PROPERTY PUBLIC classHintActive : BOOL
GET
classHintActive													:= ClassInfo[TCEVENTCLASS_HINT] <> 0;
END_GET
END_PROPERTY

PROPERTY PUBLIC classInstructionActive : BOOL
GET
classInstructionActive													:= ClassInfo[TCEVENTCLASS_INSTRUCTION] <> 0;
END_GET
END_PROPERTY

PROPERTY PUBLIC classMaintenanceActive : BOOL
GET
classMaintenanceActive													:= ClassInfo[TCEVENTCLASS_MAINTENANCE] <> 0;
END_GET
END_PROPERTY

PROPERTY PUBLIC classMessageActive : BOOL
GET
classMessageActive													:= ClassInfo[TCEVENTCLASS_MESSAGE] <> 0;
END_GET
END_PROPERTY

PROPERTY PUBLIC classNoneActive : BOOL
GET
ClassNoneActive													:= ClassInfo[TCEVENTCLASS_NONE] <> 0;
END_GET
END_PROPERTY

PROPERTY PUBLIC classParamErrorActive : BOOL
GET
ClassParamErrorActive													:= ClassInfo[TCEVENTCLASS_PARAMERROR] <> 0;
END_GET
END_PROPERTY

PROPERTY PUBLIC classStateinfoActive : BOOL
GET
ClassStateinfoActive													:= ClassInfo[TCEVENTCLASS_STATEINFO] <> 0;
END_GET
END_PROPERTY

PROPERTY PUBLIC classWarningActive : BOOL
GET
ClassWarningActive													:= ClassInfo[TCEVENTCLASS_WARNING] <> 0;
END_GET
END_PROPERTY

METHOD PUBLIC clear : BOOL //Return value = TRUE if execution finished 
VAR_INPUT
END_VAR
	MEMSET(ADR(ClassInfo),0,SIZEOF(ClassInfo));
	MEMSET(ADR(PriorityInfo),0,SIZEOF(PriorityInfo));
	NoOfQuitRequiredEvents									:= 0;	
	NoOfActiveEvents										:= 0;
	Clear													:= TRUE;
END_METHOD

{attribute 'hide'}
METHOD PUBLIC countIn : BOOL //Return value = TRUE if execution finished 
VAR_IN_OUT
	Status													:	DWORD; (*	.0 - .8 = event of <class id> is active / .15 confirm required / .16 = Level 0 , .17 = Level 1 , .18 = Level 2, ..........
																			TCEVENTCLASS_NONE			:=0,	(* No class *)
																			TCEVENTCLASS_MAINTENANCE	:=1,	(* Maintenance hint *)
																			TCEVENTCLASS_MESSAGE		:=2,	(* Message *)
																			TCEVENTCLASS_HINT			:=3,	(* Hint *)
																			TCEVENTCLASS_STATEINFO		:=4,	(* State information *)
																			TCEVENTCLASS_INSTRUCTION	:=5,	(* Instruction *)
																			TCEVENTCLASS_WARNING		:=6,	(* Warning *)
																			TCEVENTCLASS_ALARM			:=7,	(* Alarm *)
																			TCEVENTCLASS_PARAMERROR		:=8		(* Parameter error *)  *)
END_VAR
IF TestAndSet(TaskInterlockCountIn)
THEN
	IF Status.0 THEN ClassInfo[TCEVENTCLASS_NONE] 				:= ClassInfo[TCEVENTCLASS_NONE] + 1; 									
	ELSIF Status.1 THEN ClassInfo[TCEVENTCLASS_MAINTENANCE] 	:= ClassInfo[TCEVENTCLASS_MAINTENANCE] + 1; 
	ELSIF Status.2 THEN ClassInfo[TCEVENTCLASS_MESSAGE] 		:= ClassInfo[TCEVENTCLASS_MESSAGE] + 1; 	
	ELSIF Status.3 THEN ClassInfo[TCEVENTCLASS_HINT] 			:= ClassInfo[TCEVENTCLASS_HINT] + 1; 		
	ELSIF Status.4 THEN ClassInfo[TCEVENTCLASS_STATEINFO] 		:= ClassInfo[TCEVENTCLASS_STATEINFO] + 1; 	
	ELSIF Status.5 THEN ClassInfo[TCEVENTCLASS_INSTRUCTION] 	:= ClassInfo[TCEVENTCLASS_INSTRUCTION] + 1; 
	ELSIF Status.6 THEN ClassInfo[TCEVENTCLASS_WARNING] 		:= ClassInfo[TCEVENTCLASS_WARNING] + 1; 	
	ELSIF Status.7 THEN ClassInfo[TCEVENTCLASS_ALARM] 			:= ClassInfo[TCEVENTCLASS_ALARM] + 1; 		
	ELSIF Status.8 THEN ClassInfo[TCEVENTCLASS_PARAMERROR] 		:= ClassInfo[TCEVENTCLASS_PARAMERROR] + 1; 	
	END_IF
	
	IF Status.15 THEN NoOfQuitRequiredEvents 					:= NoOfQuitRequiredEvents + 1; END_IF
	
	IF status.16 THEN PriorityInfo[0]							:= PriorityInfo[0] + 1;						
	ELSIF status.17 THEN PriorityInfo[1]						:= PriorityInfo[1] + 1	;						
	ELSIF status.18 THEN PriorityInfo[2]						:= PriorityInfo[2] + 1;						
	ELSIF status.19 THEN PriorityInfo[3]						:= PriorityInfo[3] + 1;						
	ELSIF status.20 THEN PriorityInfo[4]						:= PriorityInfo[4] + 1;						
	ELSIF status.21 THEN PriorityInfo[5]						:= PriorityInfo[5] + 1;						
	ELSIF status.22 THEN PriorityInfo[6]						:= PriorityInfo[6] + 1;						
	ELSIF status.23 THEN PriorityInfo[7]						:= PriorityInfo[7] + 1	;						
	END_IF
	
	//set active flag	
	NoOfActiveEvents											:= NoOfActiveEvents + 1;
	
	status.31 													:= TRUE; 
	CountIn														:= TRUE;
	TaskInterlockCountIn										:= FALSE;
END_IF
END_METHOD

// {attribute 'hide'}
METHOD PUBLIC countOut : BOOL //Return value = TRUE if execution finished 
VAR_IN_OUT
	Status													:	DWORD; (*	.0 - .8 = event of <class id> is active / .15 confirm required / .16 = Level 0 , .17 = Level 1 , .18 = Level 2, ..........
																			TCEVENTCLASS_NONE			:=0,	(* No class *)
																			TCEVENTCLASS_MAINTENANCE	:=1,	(* Maintenance hint *)
																			TCEVENTCLASS_MESSAGE		:=2,	(* Message *)
																			TCEVENTCLASS_HINT			:=3,	(* Hint *)
																			TCEVENTCLASS_STATEINFO		:=4,	(* State information *)
																			TCEVENTCLASS_INSTRUCTION	:=5,	(* Instruction *)
																			TCEVENTCLASS_WARNING		:=6,	(* Warning *)
																			TCEVENTCLASS_ALARM			:=7,	(* Alarm *)
																			TCEVENTCLASS_PARAMERROR		:=8		(* Parameter error *)  *)
END_VAR
IF TestAndSet(TaskInterlockCountOut)
THEN
	IF Status.0 THEN ClassInfo[TCEVENTCLASS_NONE] 				:= MAX(0,ClassInfo[TCEVENTCLASS_NONE] - 1); 		
	ELSIF Status.1 THEN ClassInfo[TCEVENTCLASS_MAINTENANCE] 	:= MAX(0,ClassInfo[TCEVENTCLASS_MAINTENANCE] - 1);	
	ELSIF Status.2 THEN ClassInfo[TCEVENTCLASS_MESSAGE] 		:= MAX(0,ClassInfo[TCEVENTCLASS_MESSAGE] - 1); 		
	ELSIF Status.3 THEN ClassInfo[TCEVENTCLASS_HINT] 			:= MAX(0,ClassInfo[TCEVENTCLASS_HINT] - 1); 		
	ELSIF Status.4 THEN ClassInfo[TCEVENTCLASS_STATEINFO] 		:= MAX(0,ClassInfo[TCEVENTCLASS_STATEINFO] - 1); 	
	ELSIF Status.5 THEN ClassInfo[TCEVENTCLASS_INSTRUCTION] 	:= MAX(0,ClassInfo[TCEVENTCLASS_INSTRUCTION] - 1);	
	ELSIF Status.6 THEN ClassInfo[TCEVENTCLASS_WARNING] 		:= MAX(0,ClassInfo[TCEVENTCLASS_WARNING] - 1); 	
	ELSIF Status.7 THEN ClassInfo[TCEVENTCLASS_ALARM] 			:= MAX(0,ClassInfo[TCEVENTCLASS_ALARM] - 1); 		
	ELSIF Status.8 THEN ClassInfo[TCEVENTCLASS_PARAMERROR] 		:= MAX(0,ClassInfo[TCEVENTCLASS_PARAMERROR] - 1); 	
	END_IF
																	  
	IF Status.15 THEN NoOfQuitRequiredEvents 					:=  MAX(0,NoOfQuitRequiredEvents - 1); 	
	END_IF
																	   
	IF status.16 THEN PriorityInfo[0]							:=  MAX(0,PriorityInfo[0] - 1);						
	ELSIF status.17 THEN PriorityInfo[1]						:=  MAX(0,PriorityInfo[1] - 1);						
	ELSIF status.18 THEN PriorityInfo[2]						:=  MAX(0,PriorityInfo[2] - 1);						
	ELSIF status.19 THEN PriorityInfo[3]						:=  MAX(0,PriorityInfo[3] - 1);						
	ELSIF status.20 THEN PriorityInfo[4]						:=  MAX(0,PriorityInfo[4] - 1);						
	ELSIF status.21 THEN PriorityInfo[5]						:=  MAX(0,PriorityInfo[5] - 1);						
	ELSIF status.22 THEN PriorityInfo[6]						:=  MAX(0,PriorityInfo[6] - 1);						
	ELSIF status.23 THEN PriorityInfo[7]						:=  MAX(0,PriorityInfo[7] - 1);						
	END_IF
	
	NoOfActiveEvents											:= MAX(0,NoOfActiveEvents - 1);
	status.31													:= FALSE; //Active flag reset
	CountOut													:= TRUE;
	TaskInterlockCountOut										:= FALSE;
END_IF
END_METHOD

METHOD INTERNAL initEvent : DWORD //Return status 
VAR_IN_OUT
	SetClass								:	E_TcEventClass;
	EventConfig								:	TcEvent;
END_VAR
		(* Event Config *)
		InitEvent											:= 0;
		IF SetClass = TC2_SYSTEM.TCEVENTCLASS_NONE 				
		THEN	
			EventConfig.Class								:= SetClass;
			EventConfig.bQuitRequired						:= PARAM.EVENT_HANDLING_CONFIG.CLASS_NONE_QUIT_REQUIRED;
			InitEvent.15									:= PARAM.EVENT_HANDLING_CONFIG.CLASS_NONE_QUIT_REQUIRED;
			EventConfig.Prio								:= PARAM.EVENT_HANDLING_CONFIG.CLASS_NONE_PRIORITY;
			InitEvent										:= SETBIT32(InitEvent,TO_SINT(PARAM.EVENT_HANDLING_CONFIG.CLASS_NONE_PRIORITY) + 16);	
			InitEvent.0										:= TRUE;													
			
		ELSIF SetClass = TC2_SYSTEM.TCEVENTCLASS_MAINTENANCE 
		THEN
			EventConfig.Class								:= SetClass;
			EventConfig.bQuitRequired						:= PARAM.EVENT_HANDLING_CONFIG.CLASS_MAINTENANCE_QUIT_REQUIRED;
			InitEvent.15									:= PARAM.EVENT_HANDLING_CONFIG.CLASS_MAINTENANCE_QUIT_REQUIRED;
			EventConfig.Prio								:= PARAM.EVENT_HANDLING_CONFIG.CLASS_MAINTENANCE_PRIORITY;
			InitEvent										:= SETBIT32(InitEvent,TO_SINT(PARAM.EVENT_HANDLING_CONFIG.CLASS_MAINTENANCE_PRIORITY) + 16);
			InitEvent.1										:= TRUE;
		ELSIF SetClass = TC2_SYSTEM.TCEVENTCLASS_MESSAGE 		
		THEN
			EventConfig.Class								:= SetClass;
			EventConfig.bQuitRequired						:= PARAM.EVENT_HANDLING_CONFIG.CLASS_MESSAGE_QUIT_REQUIRED;
			InitEvent.15									:= PARAM.EVENT_HANDLING_CONFIG.CLASS_MESSAGE_QUIT_REQUIRED;
			EventConfig.Prio								:= PARAM.EVENT_HANDLING_CONFIG.CLASS_MESSAGE_PRIORITY;
			InitEvent										:= SETBIT32(InitEvent,TO_SINT(PARAM.EVENT_HANDLING_CONFIG.CLASS_MESSAGE_PRIORITY) + 16);
			InitEvent.2										:= TRUE;
		ELSIF SetClass = TC2_SYSTEM.TCEVENTCLASS_HINT 			
		THEN
			EventConfig.Class								:= SetClass;
			EventConfig.bQuitRequired						:= PARAM.EVENT_HANDLING_CONFIG.CLASS_HINT_QUIT_REQUIRED;
			InitEvent.15									:= PARAM.EVENT_HANDLING_CONFIG.CLASS_HINT_QUIT_REQUIRED;
			EventConfig.Prio								:= PARAM.EVENT_HANDLING_CONFIG.CLASS_HINT_PRIORITY;
			InitEvent										:= SETBIT32(InitEvent,TO_SINT(PARAM.EVENT_HANDLING_CONFIG.CLASS_HINT_PRIORITY) + 16);
			InitEvent.3										:= TRUE;
		ELSIF SetClass = TC2_SYSTEM.TCEVENTCLASS_STATEINFO 	
		THEN
			EventConfig.Class								:= SetClass;
			EventConfig.bQuitRequired						:= PARAM.EVENT_HANDLING_CONFIG.CLASS_STATEINFO_QUIT_REQUIRED;
			InitEvent.15									:= PARAM.EVENT_HANDLING_CONFIG.CLASS_STATEINFO_QUIT_REQUIRED;
			EventConfig.Prio								:= PARAM.EVENT_HANDLING_CONFIG.CLASS_STATEINFO_PRIORITY;
			InitEvent										:= SETBIT32(InitEvent,TO_SINT(PARAM.EVENT_HANDLING_CONFIG.CLASS_STATEINFO_PRIORITY) + 16);
			InitEvent.4										:= TRUE;
		ELSIF SetClass = TC2_SYSTEM.TCEVENTCLASS_INSTRUCTION 
		THEN
			EventConfig.Class								:= SetClass;
			EventConfig.bQuitRequired						:= PARAM.EVENT_HANDLING_CONFIG.CLASS_INSTRUCTION_QUIT_REQUIRED;
			InitEvent.15									:= PARAM.EVENT_HANDLING_CONFIG.CLASS_INSTRUCTION_QUIT_REQUIRED;
			EventConfig.Prio								:= PARAM.EVENT_HANDLING_CONFIG.CLASS_INSTRUCTION_PRIORITY;
			InitEvent										:= SETBIT32(InitEvent,TO_SINT(PARAM.EVENT_HANDLING_CONFIG.CLASS_INSTRUCTION_PRIORITY) + 16);
			InitEvent.5										:= TRUE;
		ELSIF SetClass = TC2_SYSTEM.TCEVENTCLASS_WARNING 		
		THEN
			EventConfig.Class								:= SetClass;
			EventConfig.bQuitRequired						:= PARAM.EVENT_HANDLING_CONFIG.CLASS_WARNING_QUIT_REQUIRED;
			InitEvent.15									:= PARAM.EVENT_HANDLING_CONFIG.CLASS_WARNING_QUIT_REQUIRED;
			EventConfig.Prio								:= PARAM.EVENT_HANDLING_CONFIG.CLASS_WARNING_PRIORITY;
			InitEvent										:= SETBIT32(InitEvent,TO_SINT(PARAM.EVENT_HANDLING_CONFIG.CLASS_WARNING_PRIORITY) + 16);
			InitEvent.6										:= TRUE;
		ELSIF SetClass = TC2_SYSTEM.TCEVENTCLASS_ALARM 		
		THEN
			EventConfig.Class								:= SetClass;
			EventConfig.bQuitRequired						:= PARAM.EVENT_HANDLING_CONFIG.CLASS_ALARM_QUIT_REQUIRED;
			InitEvent.15									:= PARAM.EVENT_HANDLING_CONFIG.CLASS_ALARM_QUIT_REQUIRED;
			EventConfig.Prio								:= PARAM.EVENT_HANDLING_CONFIG.CLASS_ALARM_PRIORITY;
			InitEvent										:= SETBIT32(InitEvent,TO_SINT(PARAM.EVENT_HANDLING_CONFIG.CLASS_ALARM_PRIORITY) + 16);
			InitEvent.7										:= TRUE;
		ELSIF SetClass = TC2_SYSTEM.TCEVENTCLASS_PARAMERROR 	
		THEN
			EventConfig.Class								:= SetClass;
			EventConfig.bQuitRequired						:= PARAM.EVENT_HANDLING_CONFIG.CLASS_PARAMERROR_QUIT_REQUIRED;
			InitEvent.15									:= PARAM.EVENT_HANDLING_CONFIG.CLASS_PARAMERROR_QUIT_REQUIRED;
			EventConfig.Prio								:= PARAM.EVENT_HANDLING_CONFIG.CLASS_PARAMERROR_PRIORITY;
			InitEvent										:= SETBIT32(InitEvent,TO_SINT(PARAM.EVENT_HANDLING_CONFIG.CLASS_PARAMERROR_PRIORITY) + 16);
			InitEvent.8										:= TRUE;
		ELSE 
			EventConfig.Class								:= SetClass;
			EventConfig.bQuitRequired						:= PARAM.EVENT_HANDLING_CONFIG.CLASS_ALARM_QUIT_REQUIRED;
			InitEvent.15									:= PARAM.EVENT_HANDLING_CONFIG.CLASS_ALARM_QUIT_REQUIRED;
			EventConfig.Prio								:= PARAM.EVENT_HANDLING_CONFIG.CLASS_ALARM_PRIORITY;
			InitEvent										:= SETBIT32(InitEvent,TO_SINT(PARAM.EVENT_HANDLING_CONFIG.CLASS_ALARM_PRIORITY) + 16);
			InitEvent.7										:= TRUE;
		END_IF
END_METHOD

METHOD PUBLIC isClassActive : BOOL  //Return value = TRUE if EventClass is currently active
VAR_INPUT
	TcEventClass											:	E_TcEventClass;
END_VAR
IF TcEventClass < MIN_CLASS OR TcEventClass > MAX_CLASS
THEN
	IsClassActive											:= TRUE;
ELSE
	IsClassActive											:= ClassInfo[TcEventClass] <> 0;
END_IF
END_METHOD

PROPERTY PUBLIC isConfirmReqActive : BOOL
GET
isConfirmReqActive											:= NoOfQuitRequiredEvents <> 0;
END_GET
END_PROPERTY

METHOD PUBLIC isPriorityActive : BOOL //Return value = TRUE if priority is active
VAR_INPUT
	IN														:	INT;
END_VAR
IF IN < MIN_PRIORITY OR IN > MAX_PRIORITY
THEN
	IsPriorityActive										:= TRUE;
ELSE
	IsPriorityActive										:= PriorityInfo[In] <> 0;
END_IF
END_METHOD

END_FUNCTION_BLOCK

// POUs/EventLogger/EventsWriteToLogbook
{attribute 'no_check'}
//Write new event logger messages from "ReadAdsEvent" instance into "LogBook" instance
FUNCTION_BLOCK EventsWriteToLogbook
VAR_OUTPUT CONSTANT
{attribute 'displaymode':='binary'}
	OPTION_ADD_DT_TO_MSG_STRING								:	BYTE := 2#0000_0001;
{attribute 'displaymode':='binary'}
	OPTION_ADD_CLASS_TO_MSG_STRING							:	BYTE := 2#0000_0010;
{attribute 'displaymode':='binary'}
	OPTION_ADD_SOURCE_TO_MSG_STRING							:	BYTE := 2#0000_0100;	//Default option
{attribute 'displaymode':='binary'}
	OPTION_ADD_SOURCE_ID_TO_MSG_STRING						:	BYTE := 2#0000_1000; 
{attribute 'displaymode':='binary'}
	OPTION_ADD_MSG_ID_TO_MSG_STRING							:	BYTE := 2#0001_0000;	//Default option	
{attribute 'displaymode':='binary'}
	OPTION_ADD_MSG_DT_TO_LOGBOOK_TIMESTAMP					:	BYTE := 2#0010_0000;	
{attribute 'displaymode':='binary'}
	OPTION_ADD_MSG_STATE_ID_TO_MSG_STRING					:	BYTE := 2#0100_0000;	//Add event state before text
END_VAR
VAR_INPUT
	Enable													:	BOOL	:= FALSE;	//Activate the function block
{attribute 'displaymode':='binary'}
	Options													:	BYTE 	:= OPTION_ADD_SOURCE_TO_MSG_STRING OR OPTION_ADD_MSG_ID_TO_MSG_STRING;
END_VAR                                                     
VAR_IN_OUT                                                  
	EventlogRead											:	EventlogRead;		//ReadAdsEvent instance
	LogBook													:	LogBook_wEventClass;//Logbook instance 
END_VAR                                                     
VAR_OUTPUT                                                  
	LastEventDT												:	DT;					//Date and time of last checked event
END_VAR                                                         			
VAR
(* Memory ******************************************************)
	LastEntryTimestamp										:	T_DCTIME64;			//Date of last event in this cycle
	LastEventTimestamp										:	T_DCTIME64;			//Timestamp of last added event
	ExitMarker												:	BOOL;
	MemLogbookOptions										:	BYTE;	
	MemClass												:	E_TcEventClass := TC2_SYSTEM.TCEVENTCLASS_ALARM;
	MemTimestamp											:	TIMESTRUCT;
	LenMem													:	INT;

	
(* Timer *******************************************************)

(* Trigger *****************************************************)

(* Blocks ******************************************************)

(* Error *******************************************************)

(* Dummys ******************************************************)
	i														: 	INT := 0; 
	k,j														:	INT;
	OK														:	BOOL;
END_VAR

(* Read new events and write into logbook 							*)
(********************************************************************)

(* action ***********************************************************)
IF Enable 
THEN
	IF EventlogRead.Done
	THEN //Start read events
	
		//first save Logbook settings 
		MemTimestamp										:= LogBook.Timestamp;
		MemLogbookOptions									:= LogBook.Options;		
		MemClass											:= LogBook.eClass;
	(*	LogBook.Options										:= LogBook.Options 
																AND Logbook.OPTION_WRITE_TO_ADSLOG AND Logbook.OPTION_WRITE_TO_FILE 
																AND Logbook.OPTION_ADD_TIME_TO_MSG_STRING AND Logbook.OPTION_ADD_TIME_TO_MSG_STRING ; *)
		
		//Check list for new entrys
		ExitMarker											:= FALSE;
		FOR i := EventlogRead.TotalNumberOfEvents TO EventlogRead.MIN_EVENT BY - 1  
		DO
			IF EventlogRead.Event[i].Timestamp > LastEntryTimestamp
			THEN //New entries
				IF NOT ExitMarker 
					OR //Events with event newer timestamp, exit and continue at next cycle
					EventlogRead.Event[i].Timestamp = LastEventTimestamp
				THEN //new message
					ExitMarker								:= TRUE;
					LastEventTimestamp						:= EventlogRead.Event[i].Timestamp;
										
					IF _formatMsg(EventlogRead.LangId, EventlogRead.Event[i], LogBook)
					THEN //Write message to logbook	
						Logbook();
					END_IF
					
				ELSE //add messages the next time
					EXIT; 
				END_IF
				
			ELSE //old messages
				;
			END_IF
		
		END_FOR		
		
		//Record timestamp of last event
		LastEntryTimestamp									:= LastEventTimestamp;

		//Recover old entries	
		LogBook.Options										:= MemLogbookOptions;
		LogBook.eClass										:= MemClass;
		LogBook.Timestamp									:= MemTimestamp;				
	END_IF	
END_IF

(*******************************************************************************)

METHOD PROTECTED _formatMsg : BOOL
VAR_INPUT
	Lcid													:	eLCID;
END_VAR
VAR_IN_OUT
	Event													 : EVENTLOG_READ_DATA;
	LogBook													:	LogBook_wEventClass;//Logbook instance 
END_VAR
//2020-05-30-07:06:08.436;<EventClass txt>;<Source ID>;<Event Id>;<Event state>;CoE Drive | AxisY - Remote control over fieldbus not active  	

	//Add class to log book entry
	LogBook.eClass											:= Event.eClass;	
	Logbook.Msg												:= '';
	
	//Event timestamp to logbook timestamp
	IF OPtions.5
	THEN
		LogBook.Timestamp 									:= DT_TO_SYSTEMTIME(Event.TimestampDT);			
	END_IF
	
	//add date and time
	IF Options.0
	THEN					
		LogBook.Msg											:= DT_TO_STRING(Event.TimestampDT);			
		LogBook.Msg											:= DELETE(LogBook.Msg, 3, 1); //delete DT# 
		LogBook.Msg 										:= CONCAT(LogBook.Msg,';');					
	END_IF
		
	//add event class
	IF Options.1
	THEN
		LogBook.Msg											:= CONCAT(LogBook.Msg,GetEventClassText(Event.eClass));
		LogBook.Msg 										:= CONCAT(LogBook.Msg,';');
	END_IF

	//add source id 
	IF Options.3 
	THEN
		LogBook.Msg 										:= CONCAT(LogBook.Msg,TO_STRING(Event.Sourceid));
		LogBook.Msg 										:= CONCAT(LogBook.Msg,';');		
	END_IF							
							
	//add event id 
	IF Options.4
	THEN
		LogBook.Msg 										:= CONCAT(LogBook.Msg,DWORD_TO_STRING(Event.id));
		LogBook.Msg 										:= CONCAT(LogBook.Msg,';');				
	END_IF					
	
	//add event state
	IF Options.6
	THEN
		LogBook.Msg 										:= CONCAT(LogBook.Msg,DWORD_TO_STRING(Event.State));
		LogBook.Msg 										:= CONCAT(LogBook.Msg,';');				
	END_IF					

	//add event source text
	IF Options.2
	THEN
		IF Lcid <> eLCID.CN
		THEN
			LogBook.Msg 									:= CONCAT(LogBook.Msg,WSTRING_TO_STRING(Event.Source));
			LogBook.Msg 									:= CONCAT(LogBook.Msg,' | ');	
		ELSIF NOT Options.3    
		THEN                               
			LogBook.Msg 									:= CONCAT(LogBook.Msg,CONCAT('Source Id[', UDINT_TO_STRING(Event.Sourceid)));
			LogBook.Msg 									:= CONCAT(LogBook.Msg,'] | ');								
		END_IF	
	END_IF
		
	IF Lcid <> eLCID.CN
	THEN
		LogBook.Msg											:= CONCAT(LogBook.Msg,WSTRING_TO_STRING(Event.MsgText));
	ELSE
		LogBook.Msg 										:= CONCAT(LogBook.Msg, SEL(Options.4 , CONCAT('EventId[' ,CONCAT(UDINT_TO_STRING(Event.id),'] <Unicode active>')) , '<Unicode active>'));										
	END_IF

	_formatMsg												:= TRUE;
	
(**********************************************************************************************)
END_METHOD

END_FUNCTION_BLOCK

// POUs/Logging/Logbook
{attribute 'no_check'}
//PLC Logbook for debugging, records a number of "MAX_DATA" messages with timestamp.
//The Logbook Puplisher can be used to forward messages from the logbook to several subscriber (Write into Logfile, display via EventLogger, send to Syslog Server)
//
//Parameter Timestamp needs to be updated externaly every cycle if needed
//
//Function "LogWithEventClass" is used inside
FUNCTION_BLOCK Logbook IMPLEMENTS I_Logbook                 									
VAR_OUTPUT CONSTANT     									
//Parameter
	MIN_DATA												:	INT := 1;
	MAX_DATA												:	INT := PARAM.LOGBOOK_MAX_DATA; //see library parameter to customize parameter	
                        									
//option settings to modify the message string and behavior
{attribute 'displaymode':='binary'}
	OPTION_WRITE_TO_ADSLOG									: 	BYTE :=2#0000_0100; //Write entry directly to TwinCAT logger (shown in XAE output)
{attribute 'displaymode':='binary'}
	OPTION_ADD_TIME_TO_MSG_STRING							: 	BYTE :=2#0000_1000;	//Add time stamp to message string 
{attribute 'displaymode':='binary'}
	OPTION_ADD_DATE_TO_MSG_STRING							: 	BYTE :=2#0001_0000; //Add date to message string
END_VAR                 									
VAR_INPUT               									                       		
{attribute 'displaymode':='binary'}
	Options													:	BYTE := 2#0000_0000;			(* option constants are alreay predefined, so they can accordingly be passed symbolically to the block
																								Bit 0 = 
																								Bit 1 = 
																								Bit 2 = Send to TC Ads-Logger
																								Bit 3 = Add time to message string
																								Bit 4 = Add date to message string
																								Bit 5 = 
																								Bit 6 = 
														 										Bit 7 =  								
																								*)
                        									
// InputData         	
	Timestamp												:	TIMESTRUCT; //Time stamp need to be updated cylic if it will be used
	Msg														:	STRING(PARAM.LOGBOOK_MAX_MSG_STRING_LENGHT) := ''; //Message string which will written into the DataMsg array by executing the Fb																							
END_VAR             										
VAR_OUTPUT
	Data													:	ARRAY[MIN_DATA..MAX_DATA] OF LogbookData; // Recorded messages data
	CntAddedMessages										:	INT;
END_VAR
VAR
	TaskInterlock											:	BOOL;
END_VAR

(* LogBook 									 *)
(*********************************************)

(* call method *********************************************)
	_Write(Msg);
(***********************************************************)

METHOD PROTECTED _write : BOOL
VAR_IN_OUT
	Msg														:	STRING(PARAM.LOGBOOK_MAX_MSG_STRING_LENGHT);
END_VAR
(* Write entry with every call ******************************)
IF LEN(MSG) = 0
THEN
	_Write													:= FALSE;
	RETURN;
ELSIF TestAndSet(TaskInterlock)
THEN	
	MEMMOVE(ADR(Data[MIN(MIN_DATA + 1,MAX_DATA)]), 	ADR(Data), 	SIZEOF(Data) - SIZEOF(Data[MIN_DATA]));
	
	(* Datensatz oben eintragen *)
	IF NOT Options.3 AND NOT Options.4
	THEN
		Data[MIN_DATA].Msg									:= Msg;
	ELSIF Options.3 AND Options.4              
	THEN                                                    
		Data[MIN_DATA].Msg									:= SYSTEMTIME_TO_STRING(Timestamp);
		Data[MIN_DATA].Msg									:= CONCAT(Data[MIN_DATA].Msg, ' | ');
		Data[MIN_DATA].Msg									:= CONCAT(Data[MIN_DATA].Msg, Msg);
	ELSIF Options.4                                   
	THEN                                                    
		Data[MIN_DATA].Msg									:= SYSTEMTIME_TO_STRING(Timestamp);
		Data[MIN_DATA].Msg									:=	MID(Data[MIN_DATA].Msg, 12 , 12);
		Data[MIN_DATA].Msg									:= CONCAT(Data[MIN_DATA].Msg, ' | ');
		Data[MIN_DATA].Msg									:= CONCAT(Data[MIN_DATA].Msg, Msg);
                                                            
	ELSE (* Only Date to Msg String *)                      
		Data[MIN_DATA].Msg									:= SYSTEMTIME_TO_STRING(Timestamp);
		Data[MIN_DATA].Msg									:= MID(Data[MIN_DATA].Msg, 8 , 3);
		Data[MIN_DATA].Msg									:= CONCAT(Data[MIN_DATA].Msg, ' | ');
		Data[MIN_DATA].Msg									:= CONCAT(Data[MIN_DATA].Msg, Msg);
	END_IF                                                  

	//Coyp current options from logbook into message	                                                        
	Data[MIN_DATA].Options									:= TO_WORD(Options);
		
	//Store time stamp
	Data[MIN_DATA].Timestamp								:= Timestamp;
	
	CntAddedMessages										:= MIN(MAX_DATA, CntAddedMessages + 1); 
	_Write													:= TRUE;
	TaskInterlock											:= FALSE;
END_IF

(************************************************************)
END_METHOD

METHOD PUBLIC delete : BOOL //Return value = TRUE if execution finished
VAR_INPUT
END_VAR

CntAddedMessages											:= 0;
MEMSET(ADR(Data),0,SIZEOF(Data));
delete														:= TRUE;
END_METHOD

METHOD PUBLIC getOldestMsg : BOOL //Return value TRUE = if finished successful -> new message read
VAR_IN_OUT
	data													: LogbookData;								
END_VAR
IF CntAddedMessages >= MIN_DATA AND CntAddedMessages <= MAX_DATA
	AND NOT TaskInterlock
THEN
	data													:= THIS^.Data[CntAddedMessages];
	THIS^.Data[CntAddedMessages].Options.15					:= FALSE; //New message
	CntAddedMessages										:= CntAddedMessages - 1;
	getOldestMsg											:= TRUE;
ELSE
	getOldestMsg											:= FALSE;
END_IF
END_METHOD

PROPERTY PUBLIC optAddDateToMsgText : BOOL
GET
optAddDateToMsgText := Options.4;
END_GET
SET
Options.4 := optAddDateToMsgText;
END_SET
END_PROPERTY

PROPERTY PUBLIC optAddTimeToMsgText : BOOL
GET
optAddTimeToMsgText := Options.3;
END_GET
SET
Options.3 := optAddTimeToMsgText;
END_SET
END_PROPERTY

PROPERTY Public optWiteEntryToTcAdsLogger : BOOL
GET
optWiteEntryToTcAdsLogger := Options.2;
END_GET
SET
Options.2 := optWiteEntryToTcAdsLogger;
END_SET
END_PROPERTY

{attribute 'monitoring' := 'call'}
PROPERTY PUBLIC rCntAddedMessages : Reference to INT //Reference to variable showing no of added messages (Counter will be decreased by getOldestMsg)
GET
rCntAddedMessages REF= CntAddedMessages;
END_GET
END_PROPERTY

METHOD PUBLIC readMsg : REFERENCE TO LogbookData //Return value is a REFERENCE to the by Index selected entry.  
VAR_INPUT
	Index											:	INT;						
END_VAR

readMsg													REF= THIS^.Data[LIMIT(MIN_DATA,Index,MAX_DATA)];
END_METHOD

METHOD PUBLIC write : BOOL //Return value = TRUE if execution finished
VAR_INPUT
	Msg														:	STRING(PARAM.LOGBOOK_MAX_MSG_STRING_LENGHT);
END_VAR

write														:= _Write(Msg);
IF options.2 
THEN
	write 													:= write AND 0 = adsLogHint(Msg, '');
END_IF
END_METHOD

END_FUNCTION_BLOCK

// POUs/Logging/I_Logbook
INTERFACE I_Logbook Extends __System.IQueryInterface

METHOD PUBLIC delete : BOOL //Return value = TRUE if execution finished
VAR_INPUT
END_VAR
END_METHOD

METHOD PUBLIC getOldestMsg : BOOL //Return value TRUE = if finished successful -> new message flag of entry will be reset
VAR_IN_OUT
	data													: LogbookData;								
END_VAR
END_METHOD

{attribute 'monitoring' := 'call'}
PROPERTY PUBLIC rCntAddedMessages : Reference to INT
GET
END_GET
END_PROPERTY

METHOD PUBLIC readMsg : REFERENCE TO LogbookData //Return value is a REFERENCE to the by Index selected entry.  
VAR_INPUT
	Index											:	INT;						
END_VAR
END_METHOD

METHOD PUBLIC write : BOOL //Return value = TRUE if execution finished
VAR_INPUT
	Msg														:	STRING(PARAM.LOGBOOK_MAX_MSG_STRING_LENGHT);
END_VAR
END_METHOD

END_INTERFACE

// POUs/Logging/Logbook_wEventClass
{attribute 'no_check'}
FUNCTION_BLOCK Logbook_wEventClass EXTENDS Logbook             									
VAR_OUTPUT CONSTANT     									
END_VAR                 									
VAR_INPUT               									                       		
	eClass													:	E_TcEventClass := TC2_SYSTEM.TCEVENTCLASS_NONE; //Possible event class for the entry																							
END_VAR             										
VAR_OUTPUT
END_VAR
VAR

END_VAR

(* LogBook 									 *)
(*********************************************)

(* call method *********************************************)
	Write(Msg);
(***********************************************************)

METHOD PUBLIC getClassFromOption : E_TcEventClass
VAR_INPUT
	Msgidx														:	INT;
END_VAR
IF Msgidx >= MIN_DATA AND Msgidx <= MAX_DATA
THEN
	GetClassFromOption.0 										:= Data[Msgidx].Options.8;
	GetClassFromOption.1 										:= Data[Msgidx].Options.9;
	GetClassFromOption.2 										:= Data[Msgidx].Options.10;
	GetClassFromOption.3 										:= Data[Msgidx].Options.11;
ELSE
	GetClassFromoption 											:= TCEVENTCLASS_ALARM;
END_IF
END_METHOD

METHOD PUBLIC write : BOOL //Return value = TRUE if execution finished
VAR_INPUT
	Msg														:	STRING(PARAM.LOGBOOK_MAX_MSG_STRING_LENGHT);
END_VAR

IF _Write(Msg)
THEN
	//Store class as integer in logbook options
	Data[MIN_DATA].Options.8								:= eClass.0;
	Data[MIN_DATA].Options.9								:= eClass.1; 
	Data[MIN_DATA].Options.10								:= eClass.2; 
	Data[MIN_DATA].Options.11								:= eClass.3;	
	write													:= TRUE;											
	
	IF options.2 
	THEN
		write												:= 0= adsLogwTcEventClass(Msg, eClass);
	END_IF
END_IF
END_METHOD

METHOD PUBLIC writeWithClass : BOOL //Return value = TRUE if execution finished
VAR_INPUT
	Msg														:	STRING(PARAM.LOGBOOK_MAX_MSG_STRING_LENGHT);
	Class													:	E_TcEventClass := TC2_SYSTEM.TCEVENTCLASS_NONE;
END_VAR
IF _Write(Msg)
THEN
	//Store class as integer in logbook options
	Data[MIN_DATA].Options.8								:= Class.0;
	Data[MIN_DATA].Options.9								:= Class.1; 
	Data[MIN_DATA].Options.10								:= Class.2; 
	Data[MIN_DATA].Options.11								:= Class.3;	
	writeWithClass											:= TRUE;
	IF options.2 
	THEN
		writeWithClass 										:= 0 = adsLogwTcEventClass(Msg, Class);
	END_IF
END_IF
END_METHOD

END_FUNCTION_BLOCK

// POUs/Logging/adsLogwTcEventClass
{attribute 'no_check' := ''}
//Writing string as hint message into the TwinCAT ams logger and windows event log with a Lreal argument
//Please see Beckhoff information system "ADSLOGLREAL" for detailed information.
//Intention of this function is to use the handy ADSLOGxxxx without the annoying msgCtrlMask as a parameter :-)  
//Function "EventHandlingGetClassLevel" is used inside
FUNCTION adsLogwTcEventClass : DINT
VAR_INPUT               											
	MsgFmtStr												:	T_MaxString;
(*	dintArg													:	DINT; *) 
(*	strArg													:	T_MaxString; *)
(*	realArg													:	LREAL; *)
	TcEventClass											:	E_TcEventClass; 
END_VAR
VAR
	msgCtrlMask												:	DWORD; (* 	ADSLOG_MSGTYPE_HINT Meldungstyp ist Hinweis.
																				ADSLOG_MSGTYPE_WARN Meldungstyp ist Warnung.  
																				ADSLOG_MSGTYPE_ERROR Meldungstyp ist Fehler.  
																				ADSLOG_MSGTYPE_LOG Meldung wird in das Logbuch geschrieben.  
																				ADSLOG_MSGTYPE_MSGBOX Meldung wird in einer Messagebox ausgegeben.  
																				ADSLOG_MSGTYPE_RESOURCE Meldung wird aus einer Ressource-Datei geholt. (wird momentan nicht  unterstützt)  
																				ADSLOG_MSGTYPE_STRING 	Meldung ist direkt angegebener String (default).  *)	
END_VAR

(* create fixed message ctrl mask **********************************)
	CASE GetEventClassPriority(tcEventClass) OF 
	0:	msgCtrlMask											:= ADSLOG_MSGTYPE_HINT;
	1:	msgCtrlMask											:= ADSLOG_MSGTYPE_WARN;
	ELSE
		msgCtrlMask											:= ADSLOG_MSGTYPE_ERROR;
	END_CASE

	msgCtrlMask												:= ADSLOG_MSGTYPE_STRING OR msgCtrlMask OR ADSLOG_MSGTYPE_LOG;

(* write string which includes a floating-number ******************)
	adsLogwTcEventClass 										:= ADSLOGLREAL(msgCtrlMask, msgFmtStr, 0.0);
	
(* write string which includes a DINT-number *******************)
(*	LogWithEventClass 										:= ADSLOGDINT(msgCtrlMask, msgFmtStr, dintArg); *)

(* write string which includes an other string e.g. 'hallo: %s what's up' ***************)
(*	LogWithEventClass 										:= ADSLOGSTR(msgCtrlMask, msgFmtStr,msgCtrlMaskstrArg); *)

(*****************************************************)

END_FUNCTION

// POUs/EventLogger/getEventClassPriority
{attribute 'no_check'}
//Returns configured level to corresponding event class (see library Param) 
FUNCTION getEventClassPriority : UINT
VAR_INPUT
	TcEventClass											:	E_TcEventClass;
END_VAR
VAR
END_VAR

	CASE tcEventClass OF
	Tc2_System.TCEVENTCLASS_NONE:			GetEventClassPriority	:= PARAM.EVENT_HANDLING_CONFIG.CLASS_NONE_PRIORITY;	
	Tc2_System.TCEVENTCLASS_MAINTENANCE:	GetEventClassPriority	:= PARAM.EVENT_HANDLING_CONFIG.CLASS_MAINTENANCE_PRIORITY;		
	Tc2_System.TCEVENTCLASS_MESSAGE:		GetEventClassPriority	:= PARAM.EVENT_HANDLING_CONFIG.CLASS_MESSAGE_PRIORITY;			
	Tc2_System.TCEVENTCLASS_HINT:			GetEventClassPriority	:= PARAM.EVENT_HANDLING_CONFIG.CLASS_HINT_PRIORITY;	
	Tc2_System.TCEVENTCLASS_STATEINFO:		GetEventClassPriority	:= PARAM.EVENT_HANDLING_CONFIG.CLASS_STATEINFO_PRIORITY;	
	Tc2_System.TCEVENTCLASS_INSTRUCTION:	GetEventClassPriority	:= PARAM.EVENT_HANDLING_CONFIG.CLASS_INSTRUCTION_PRIORITY;	
	Tc2_System.TCEVENTCLASS_WARNING:		GetEventClassPriority	:= PARAM.EVENT_HANDLING_CONFIG.CLASS_WARNING_PRIORITY;	
	Tc2_System.TCEVENTCLASS_ALARM:			GetEventClassPriority	:= PARAM.EVENT_HANDLING_CONFIG.CLASS_ALARM_PRIORITY;	
	Tc2_System.TCEVENTCLASS_PARAMERROR:		GetEventClassPriority	:= PARAM.EVENT_HANDLING_CONFIG.CLASS_PARAMERROR_PRIORITY;		
	ELSE
		GetEventClassPriority										:= PARAM.EVENT_HANDLING_CONFIG.CLASS_ALARM_PRIORITY;
	END_CASE

END_FUNCTION

// POUs/EventLogger/getEventClassText
//Returns event class in english and upper case letters 
FUNCTION getEventClassText : STRING(12)
VAR_INPUT
	TcEventClass													: E_TcEventClass;
END_VAR
VAR
END_VAR

CASE TcEventClass OF
TC2_SYSTEM.TCEVENTCLASS_NONE		: GetEventClassText 	:= 'NONE';	
TC2_SYSTEM.TCEVENTCLASS_MESSAGE		: GetEventClassText 	:= 'MESSAGE';	
TC2_SYSTEM.TCEVENTCLASS_HINT		: GetEventClassText 	:= 'HINT';	
TC2_SYSTEM.TCEVENTCLASS_STATEINFO	: GetEventClassText 	:= 'STATEINFO';	
TC2_SYSTEM.TCEVENTCLASS_INSTRUCTION	: GetEventClassText 	:= 'INSTRUCTION';			 										
TC2_SYSTEM.TCEVENTCLASS_WARNING		: GetEventClassText 	:= 'WARNING';	
TC2_SYSTEM.TCEVENTCLASS_MAINTENANCE	: GetEventClassText 	:= 'MAINTENANCE';		 														
TC2_SYSTEM.TCEVENTCLASS_ALARM		: GetEventClassText 	:= 'ALARM';	
TC2_SYSTEM.TCEVENTCLASS_PARAMERROR	: GetEventClassText 	:= 'PARAMERROR';		
ELSE
	GetEventClassText										:= 'UNKNOWN';
END_CASE

END_FUNCTION

// POUs/Fieldbus/CANopen/CANopenMasterDiag
{attribute 'no_check'}
//EL6751 CanOpen Master via EtherCAT
FUNCTION_BLOCK CANopenMasterDiag                   								
VAR_INPUT                   								
	Enable													:	BOOL := TRUE;		//FB will be processed as long as enable is TRUE 
	ConfirmTrig												:	BOOL;               //Resets error with rising edge        								
	SourceId												: 	UDINT :=  103010; 	//Multisource id 
(* Components *)            								
	IO														:	CanOpenMasterIO;
END_VAR                     								
VAR_OUTPUT                  								
	MasterOK												:	BOOL;				//TRUE when Master Device is OK
	FieldOK													:	BOOL;				//TRUE when Field Devices (Slaves) are OK
END_VAR                     	
VAR
(* internal used variables ***********************************************)
	Rx_ErrorCounter											:	USINT := 0;
	Tx_ErrorCounter											: 	USINT := 0;

(* events *********************************************************)
	Event													:	EventHandlingGrp10 := (AutoConfirm	:= FALSE);
	
(* Dummys **********************************************************)
	i														:	INT ;

END_VAR

	(* CanOpen Master Diag Ctrl 					*)
	(************************************************)

(* Work IO *************************************************)
	IO();

(* Events **************************************************)
	IF Event.no[1].Text1 <> IO.Name OR Event.no[1].Text1 <> ''
	THEN
		FOR i := Event.MIN_EVENT TO Event.MAX_EVENT DO
			Event.no[1].Text1								:= IO.Name;
		END_FOR	
	END_IF

(* 
  Bit 0: CAN-Controller is in BUS-OFF
  Bit 1: CAN-Controller warning limit reached
  Bit 2: Rx-Queue overrun
  Bit 3: Hi-Prio Tx-Queue overrun
  Bit 4: Lo-Prio Tx-Queue overrun
  Bit 5: CAN-Send Error
*)
	Event.no[1].Flag 										:= IO.CanState.0;
	Event.no[2].Flag 										:= IO.CanState.1;
	Event.no[3].Flag 										:= IO.CanState.2;   
	Event.no[4].Flag 										:= IO.CanState.3;   
	Event.no[5].Flag 										:= IO.CanState.4; 	
	Event.no[6].Flag 										:= IO.CanState.5;
	
	IF Rx_ErrorCounter <> IO.RXErrorCounter 
	THEN
		Rx_ErrorCounter 									:= IO.RXErrorCounter;
		Event.no[7].Text1 									:= USINT_TO_STRING(Rx_ErrorCounter);
		Event.no[7].Flag									:= TRUE;		
	ELSIF ConfirmTrig
	THEN
		Event.no[7].Flag									:= FALSE;
	END_IF

	IF Tx_ErrorCounter <> IO.TxErrorCounter
	THEN
		Tx_ErrorCounter 									:= IO.TXErrorCounter;
		Event.no[8].Text1 									:= USINT_TO_STRING(Tx_ErrorCounter);
		Event.no[8].Flag									:= TRUE;		
	ELSIF ConfirmTrig
	THEN
		Event.no[8].Flag 									:= FALSE;
	END_IF	

	Event.no[9].Flag 										:= FALSE;
	Event.no[10].Flag 										:= FALSE;	
	
	Event(
		ConfirmTrig := ConfirmTrig,
		Disable		:= NOT Enable,
		SourceId	:= SourceId);
	

(*******************************************************************************************)

END_FUNCTION_BLOCK

// POUs/Fieldbus/CANopen/CANopenMasterIO
{attribute 'no_check'}
//EL6751 CanOpen Master IOs
FUNCTION_BLOCK CANopenMasterIO
VAR_INPUT
END_VAR
VAR_OUTPUT
(* Inputs *)
	AdsAddr											AT %I*	:	AMSADDR;	//Terminal AMS Net Addr.
	AmsNetIdStr												:	T_AmsNetId;	//AmsNetId String
	EcMasterDevId									AT %I*	: 	UINT; 		//Map to EtherCAT Master DevId
	
	Error											AT %I*	:	USINT;		//Rising edge of Error informs that an error occurred during the execution of the Function Block 
	CanState										AT %I*	:	UINT;		//State of Can Bus
	RXErrorCounter									AT %I*	:	USINT;		//Rx error counter of the CAN controller
	TxErrorCounter									AT %I*	:	USINT;		//Tx error counter of the CAN controller
	DiagFlag										AT %I*	:	BOOL;		//Diag Flag of the last configured CANopen slave
	Name													:	STRING(30) := '';
END_VAR                         					
VAR_OUTPUT CONSTANT
END_VAR
VAR
	IOF_GetBoxNameByAddr									:	IOF_GetBoxNameByAddr := (NETID := '', TMOUT := DEFAULT_ADS_TIMEOUT);
END_VAR

(* CANopen master IO diag										             	 		*)
(********************************************************************************)

(* Get name ******************************************************************************)
IF Name = ''
	AND AdsAddr.port <> 0 AND EcMasterDevId <> 0
	OR IOF_GetBoxNameByAddr.BUSY
	OR IOF_GetBoxNameByAddr.START
THEN
	AmsNetIdStr												:= F_CreateAmsNetId(nIds := AdsAddr.netId);
		
	IOF_GetBoxNameByAddr(
		NETID		:=  , (* Local *)
		DEVICEID	:= UINT_TO_UDINT(EcMasterDevId) ,
		BOXADDR		:= AdsAddr.port ,
		START		:= Name = '' AND NOT IOF_GetBoxNameByAddr.BUSY,
		TMOUT		:= ,
		BOXNAME		=> name);
END_IF
(********************************************************************************)

PROPERTY PUBLIC setName : STRING //Set name if device is not an Ethercat terminal
SET
Name := SetName;
END_SET
END_PROPERTY

END_FUNCTION_BLOCK

// POUs/Fieldbus/EAP/EAP_DEVICE_IO
{attribute 'no_check'}
FUNCTION_BLOCK EAP_DEVICE_IO 
VAR_OUTPUT CONSTANT
END_VAR
VAR_INPUT
	{attribute 'displaymode':='hex'}
	DevCtrl				AT %Q*:	UINT;
END_VAR		
VAR_OUTPUT	
	{attribute 'displaymode':='hex'}
	DevState			AT %I*:	UINT;
	
	LinkError				:	BOOL; //0x0001 = Link error
	IOLockedAfterLinkErr	:	BOOL; //0x0002 = I/O locked after link error (I/O reset required)
	OutOfSendResources		:	BOOL; //0x0010 = Out of send resources (I/O reset required)
	WatchdogTriggered		:	BOOL; //0x0020 = Watchdog triggered
	EthMiniportNotFound		:	BOOL; //0x0040 = Ethernet driver (miniport) not found
	ResetActive				:	BOOL; //0x0080 = I/O reset active
END_VAR
VAR
END_VAR

	(* IOs 									*)
	(****************************************)

(* Read status *****************************************)
	LinkError				:= DevState.0;
	IOLockedAfterLinkErr	:= DevState.1;
	
	OutOfSendResources		:= DevState.4;
	WatchdogTriggered		:= DevState.5;
	EthMiniportNotFound		:= DevState.6;
	ResetActive				:= DevState.7;
	
(*******************************************************)

PROPERTY PUBLIC resetRequired : bool
GET
resetRequired := IOLockedAfterLinkErr or OutOfSendResources;
END_GET
END_PROPERTY

END_FUNCTION_BLOCK

// POUs/Fieldbus/EAP/EAP_PUB_SUB_IO
{attribute 'no_check'}
//Publisher/Subscriber IOs
FUNCTION_BLOCK EAP_PUB_SUB_IO 
VAR_OUTPUT CONSTANT
END_VAR
VAR_INPUT
	{attribute 'displaymode':='hex'}
	FrameCtrl									AT %Q*:	UINT;
END_VAR		
VAR_OUTPUT	
	{attribute 'displaymode':='hex'}
	FrameState									AT %I*:	UINT;
	
	NotSentFrameSkipped								: Bool;
	ErrorFrameOversized								: Bool;
	SubscriberMissing								: Bool;
END_VAR
VAR
END_VAR

	(* IOs 									*)
	(****************************************)

(* Read status *****************************************)
	NotSentFrameSkipped						:= FrameState.0;
	ErrorFrameOversized						:= FrameState.1;
	SubscriberMissing						:= FrameState.2;

(*******************************************************)

PROPERTY PUBLIC disableSending : BOOL
GET
disableSending		:= FrameCtrl.1;
END_GET
SET
FrameCtrl.1				:= disableSending;
END_SET
END_PROPERTY

PROPERTY PUBLIC removeDestMacFromARPCache : BOOL
GET
RemoveDestMacFromARPCache		:= FrameCtrl.1;
END_GET
SET
FrameCtrl.1				:= RemoveDestMacFromARPCache;
END_SET
END_PROPERTY

END_FUNCTION_BLOCK

// POUs/Fieldbus/EAP/EAP_PUB_VAR
{attribute 'no_check'}
//Default IOs of a Publisher network variable 
FUNCTION_BLOCK EAP_PUB_VAR 
VAR_OUTPUT CONSTANT
END_VAR
VAR_INPUT
	VarId						AT %Q*:	UINT;
	{attribute 'displaymode':='hex'}
	VarCtrl						AT %Q*:	UINT;
END_VAR		
VAR_OUTPUT	
	{attribute 'displaymode':='hex'}
	VarState					AT %I*:	UINT;
	
	NotSentVarSkipped					:	BOOL;
END_VAR
VAR
END_VAR

	(* IOs 									*)
	(****************************************)

NotSentVarSkipped							:= VarState.0;

PROPERTY PUBLIC disablePublishing : BOOL
GET
disablePublishing		:= VarCtrl.0;
END_GET
SET
VarCtrl.0				:= disablePublishing;
END_SET
END_PROPERTY

END_FUNCTION_BLOCK

// POUs/Fieldbus/EAP/EAP_SUB_VAR
{attribute 'no_check'}
//Default IOs of a Subscriber network variable 
FUNCTION_BLOCK EAP_SUB_VAR 
VAR_OUTPUT CONSTANT
END_VAR
VAR_INPUT
	VarId					AT %Q*:	UINT;	
	{attribute 'displaymode':='hex'}
	VarCtrl					AT %Q*:	UINT;
END_VAR		
VAR_OUTPUT	
	{attribute 'displaymode':='hex'}
	VarState				AT %I*:	UINT;
	Quality					AT %I*:	UINT;//Duration the variable is not refreshed (in 100µs/0.1ms)	
	CycleIndex				AT %I*:	UINT;//Incremented each publisher cycle
	
	QualityLT					 : LTIME;
	QualityLTMax				 : LTIME;
	
	InvalidHashValueReceived		:	BOOL;
	InvalidVarLengthReceived		:	bool;
END_VAR
VAR
END_VAR

	(* IOs 									*)
	(****************************************)

	QualityLT 								:= TO_LTIME(quality * 100000); //Quality in 100µs to ms
	IF QualityLT > QualityLTMax
	THEN
		QualityLTMax						:= QualityLT;
	END_IF
	
	InvalidHashValueReceived				:= VarState.0;
	InvalidVarLengthReceived				:= VarState.1;

PROPERTY PUBLIC ignoreHashValue : BOOL
GET
ignoreHashValue		:= VarCtrl.0;
END_GET
SET
VarCtrl.0				:= ignoreHashValue;
END_SET
END_PROPERTY

END_FUNCTION_BLOCK

// POUs/Fieldbus/EtherCAT/_Components/EcMasterIO
{attribute 'no_check'}
//EtherCAT Master Device IOs
FUNCTION_BLOCK EcMasterIO
VAR CONSTANT
	DELAY_LINK_OK											:	TIME := T#1S;
END_VAR
VAR_OUTPUT CONSTANT
	MIN_FRAMES												:	INT := 0;
	MAX_FRAMES												:	INT := PARAM.ETHERCAT_MASTER_DEV_IO_MAX_FRAMES; 
END_VAR	            							
VAR_INPUT           							                 							
(* Outputs *)       							
	FrmCtrl											AT %Q*	:	ARRAY [MIN_FRAMES..MAX_FRAMES] OF UINT;	//Link to EtherCAT Master "FrmCtrlXXX" under Outputs, e.g. 0x0001 = prevent 1. EtherCAT command from sending (request NOP)
	FrmWcCtrl										AT %Q*	:	ARRAY [MIN_FRAMES..MAX_FRAMES] OF UINT;	//Link to EtherCAT Master "FrmWcCtrlXXX" under Outputs, e.g. 0x0001 = copy data with wrong working counter of 1. EtherCAT command
	                							
	DevCtrl											AT %Q*	:	UINT := 0; //Link to EtherCAT Master "DevCtrl" under Outputs
END_VAR             							
VAR_OUTPUT          							    
	Name													:	STRING(30) := '';
								
	LinkOK_PortA											:	BOOL;		//TRUE when link is OK on port A
	LinkOK_PortB											:	BOOL;		//TRUE when link is OK on port B - Redundancy port 

	{attribute 'displaymode':='hex'}  
	DevState										AT %I*	:	UINT; (*	Link to EtherCAT Master "DevState" under Inputs,
																				0x0001 = Link error
																				0x0002 = I/O locked after link error (I/O reset required)
																				0x0004 = Link error (redundancy adapter)
																				0x0008 = Missing one frame (redundancy mode)
																				0x0010 = Out of send resources (I/O reset required)
																				0x0020 = Watchdog triggered
																				0x0040 = Ethernet driver (miniport) not found
																				0x0080 = I/O reset active
																				0x0100 = At least one device in 'INIT' state
																				0x0200 = At least one device in 'PRE-OP' state
																				0x0400 = At least one device in 'SAFE-OP' state
																				0x0800 = At least one device indicates an error state
																				0x1000 = DC not in sync *)
	DevStateText											:	T_MAXSTRING;		//shows string of device state
	DevStateBits											:	EC_MASTER_DEVICE_STATE;
	DevStateChanged											:	BOOL; //TRUE if device state changed compared to previous cylce								
   	ResetRequired											:	BOOL;		//TRUE when a reset is requested
	MinOneSlaveNotInOP										:	BOOL;		//TRUE when at least one slave is available but not in OP state
    
	NoOfFrames												:	INT;		//No of frames configured
	FrmState										AT %I*	:	ARRAY [MIN_FRAMES..MAX_FRAMES] OF UINT;	//Link to EtherCAT Master "FrmStateXXX" under Inputs, e.g. 0x0001 = 1. EtherCAT command not sent (NOP requested)
	FrmWcState										AT %I*	:	ARRAY [MIN_FRAMES..MAX_FRAMES] OF UINT;	//Link to EtherCAT Master "FrmWcStateXXX" under Inputs, e.g. 0x0001 = wrong working counter of 1. EtherCAT command received
	FrmInputToggle									AT %I*	:	ARRAY [MIN_FRAMES..MAX_FRAMES] OF UINT;	//Link to EtherCAT Master "FrmInputToggleXXX" under Inputs, e.g. 0x0001 = Toggle Bit: 1. EtherCAT command received new inputs
	AllFramesMissing										:	BOOL;		//TRUE if all frames are missing 
	FramesWCState											:	BOOL;		//TRUE if WC state in at least one frame is <> 0
	FramesWcStateChanged									:	BOOL;		//TRUE if WC state of at least one frame changed compared to previous cylce	
	
	SlaveCount										AT %I*	:	UINT;	//Link to EtherCAT Master "SlaveCount" under Inputs, show actual numer of slaves 
	SlaveCount2										AT %I*	:	UINT;	//Link to EtherCAT Master "SlaveCount2" under Inputs, show actual numer of slaves in redunance mode
	SlaveCountTotal											:	UINT; 		//Slave count 1 and 2
	RedundanceActive										:	BOOL;		//Redundance active 		
            																				                    	
(* InfoData *)      	
	ChangeCount										AT %I*	:	UINT;					//Link to EtherCAT Master "ChangeCount" under InfoData, shows how often the image of content has changed
	DevId											AT %I*	:	UINT;					//Link to EtherCAT Master "DevId" under InfoData 
 	AmsNetId										AT %I*	:	ARRAY[0..5] OF BYTE; 	//Link to EtherCAT Master "AmsNetId" under InfoData
	AmsNetIdStr												:	T_AmsNetId;	//EtherCAT Master AmsNetId in string format
	CfgSlaveCount									AT %I*	:	UINT;					////Link to EtherCAT Master "CfgSlaveCount" under InfoData, reports configured no of EtherCAT slaves
         
(* DC timestamp *)
	DCTime													:	T_DCTIME64; // RealtimeTick in DC time 64, refreshed once per cycle*)             					
						
END_VAR

VAR
	MemDevState												:	UINT := 9999;	
	MemFrmWcState											:	ARRAY [MIN_FRAMES..MAX_FRAMES] OF UINT;	

	IOF_GetDeviceName										: 	IOF_GetDeviceName := (TMOUT	:= DEFAULT_ADS_TIMEOUT);
	EcMasterFrameCount										:	FB_EcMasterFrameCount := (tTimeout	:= DEFAULT_ADS_TIMEOUT);
	TON_LinkOK_PortA										:	TON := (PT := DELAY_LINK_OK);
	TON_LinkOK_PortB										:	TON := (PT := DELAY_LINK_OK);
	i														:	INT;
END_VAR

(* EcMaster IOs *)
DevStateChanged												:= DevState <> MemDevState;
IF DevStateChanged
THEN
	DevStateBits.NoError									:= DevState = 0;
	DevStateBits.LinkError 									:= DevState.0;
	DevStateBits.IOLockedAfterLinkError	    				:= DevState.1;
	DevStateBits.LinkErrorRedMode							:= DevState.2;
	DevStateBits.MissingOneFrmInRedMode     				:= DevState.3;
	DevStateBits.OutOfSendResources         				:= DevState.4;
	DevStateBits.WatchdogTriggered 		    				:= DevState.5;
	DevStateBits.EthernetDriverNotFound 					:= DevState.6;
	DevStateBits.IOResetActive 			    				:= DevState.7;
	DevStateBits.AtLeastOneSlaveInINIT      				:= DevState.8;
	DevStateBits.AtLeastOneSlaveInPREOP     				:= DevState.9;
	DevStateBits.AtLeastOneSlaveInSAFEOP    				:= DevState.10;
	DevStateBits.AtLeastOneSlaveInERROR     				:= DevState.11;																
	DevStateBits.DcNotInSync 		        				:= DevState.12;
	DevStateText 											:= F_ConvMasterDevStateToString(DevState);
	ResetRequired 											:= DevStateBits.IOLockedAfterLinkError OR DevStateBits.OutOfSendResources;
	MinOneSlaveNotInOP										:= DevStateBits.AtLeastOneSlaveInINIT OR DevStateBits.AtLeastOneSlaveInPREOP OR  DevStateBits.AtLeastOneSlaveInSAFEOP OR DevStateBits.AtLeastOneSlaveInERROR;
	MemDevState												:= DevState;
END_IF

RedundanceActive 											:= SlaveCount2 <> 0 AND SlaveCount <> 0;
SlaveCountTotal												:= SlaveCount2 + SlaveCount;

TON_LinkOK_PortA(IN:= NOT DevStateBits.LinkError 		, Q=> LinkOK_PortA );
TON_LinkOK_PortB(IN:= NOT DevStateBits.LinkErrorRedMode	, Q=> LinkOK_PortB );

AllFramesMissing 											:= TRUE;
FramesWCState												:= FALSE;	
FramesWcStateChanged										:= FALSE;
FOR i := MIN_FRAMES TO LIMIT(0,NoOfFrames -1, MAX_FRAMES) DO
	IF FrmWcState[i] <> 0 THEN
		FramesWCState										:= TRUE;
		IF FrmWcState[i].15 OR FrmWcState[i] = 16#7FFF THEN
			;
		ELSE
			AllFramesMissing 								:= FALSE;
		END_IF
	ELSE
		AllFramesMissing 									:= FALSE;
	END_IF
	
	IF MemFrmWcState[i] <> FrmWcState[i] 
	THEN
		FramesWcStateChanged								:= TRUE;
		MemFrmWcState[i]									:= FrmWcState[i]; 
	END_IF
END_FOR

//Get DC time 
DCTime														:= F_GetCurDcTickTime64();

(* Get Master Name *)
IF Name = ''
	AND DevId <> 0
	OR IOF_GetDeviceName.BUSY
	OR IOF_GetDeviceName.START
THEN
	AmsNetIdStr 											:= F_CreateAmsNetId(nIds := AmsNetId);
	IOF_GetDeviceName(
		NETID		:= '',
		DEVICEID	:= DevId,
		START		:= Name = '' AND NOT IOF_GetDeviceName.BUSY,
		TMOUT		:= ,
		BUSY		=> ,
		ERR			=> ,
		ERRID		=> ,
		DEVICENAME=> name);
END_IF

//No of config slaves 
IF EcMasterFrameCount.nFrames = 0
	AND DevId <> 0 
	OR EcMasterFrameCount.bBusy
	OR EcMasterFrameCount.bExecute
THEN
	EcMasterFrameCount(
		sNetId	:= AmsNetIdStr, 
		bExecute:= EcMasterFrameCount.nFrames = 0 AND NOT EcMasterFrameCount.bBusy, 
		tTimeout:= , 
		bBusy=> , 
		bError=> , 
		nErrId=> , 
		nFrames=> );
	NoOfFrames												:= TO_INT(EcMasterFrameCount.nFrames);
END_IF

(********************************************************************************************************)

END_FUNCTION_BLOCK

// POUs/Fieldbus/EtherCAT/_Components/EcMasterSupervisor
{attribute 'no_check'}
// Set state of EtherCAT Master(ReqState <> 0) or read state and frame statistic 
// The FB will automatically perform a device reset if the requested state cannot be reached within the TIMEOUT_SET_STATE period
// In addition via options is possible to clear the frame statistic while set or read the Master state
FUNCTION_BLOCK EcMasterSupervisor EXTENDS FbBase
VAR CONSTANT
	TIMEOUT_SET_STATE										:	TIME := T#15S;
END_VAR
VAR_OUTPUT CONSTANT
{attribute 'displaymode':='binary'}
	OPTION_CLEAR_CRC_ERROR_COUNTER							:	BYTE := 2#0000_0001; //delete the CRC error counters of all EtherCAT slaves
{attribute 'displaymode':='binary'}
	OPTION_CLEAR_LOST_FRAMES_COUNTER						:	BYTE := 2#0000_0010; //delete the CRC error counters of all EtherCAT slaves.
{attribute 'displaymode':='binary'}	
	OPTION_CLEAR_TXRX_ERROR_COUNTER							:	BYTE := 2#0000_0100; //delete the error counters of the miniport driver of the network card
{attribute 'displaymode':='binary'}	
	OPTION_FORCE_DEVICE_RESET								:	BYTE := 2#1000_0000; //Force to execute a device reset prior to set state
END_VAR
VAR_INPUT
	AmsNetId												:	T_AmsNetId;	
	DevId													:	WORD;		//Id of mentioned device
{attribute 'displaymode':='binary'}
	Options													:	BYTE := 0; //Select	which error counter should be deleted 
{attribute 'displaymode':='hex'}
	ReqState												:	WORD := 0; (* 	Requested EtherCAT state 
																				EC_DEVICE_STATE_INIT		:BYTE 	:=16#01;
																				EC_DEVICE_STATE_PREOP		:BYTE 	:=16#02;
																				EC_DEVICE_STATE_BOOTSTRAP	:BYTE 	:=16#03;
																				EC_DEVICE_STATE_SAFEOP		:BYTE 	:=16#04;
																				EC_DEVICE_STATE_OP			:BYTE 	:=16#08; *)

END_VAR                     							
VAR_OUTPUT                  										
	ReqStateOK												:	BOOL;	//Requested EtherCAT state OK
{attribute 'displaymode':='hex'}
	CurrState												:	WORD;	//Shows current EtherCAT state
	StateText												:	STRING;	//EtherCAT State as text
	DevResetDone											:	BOOL;	//Device was reseted
//Frames statistic
    LostFrames 												: 	UDINT; //Current number of lost or invalid cyclic frames
    FramesPerSecond 										: 	LREAL; //Current number of cyclic frames per second
    LostQueuedFrames 										: 	UDINT; //Current number of lost or invalid queued (acyclic) frames
    QueuedFramesPerSecond 									: 	LREAL; //Returns the current number of queued (acyclic) frames per second
	
	ErrorText												:	STRING;
END_VAR                     								
VAR                         								
	ErrCntreset													:	INT;
	TON_TimeoutSetStatus									:	TON;
	TON_GetStateTrig										:	TON;
	MemReqState												:	WORD;

	SetMasterState											:	FB_EcSetMasterState := (tTimeout := DEFAULT_ADS_TIMEOUT);
	GetMasterState											:	FB_EcGetMasterState := (tTimeout := DEFAULT_ADS_TIMEOUT);
	ReadMasterFrameStatistic								:	FB_EcMasterFrameStatistic:= (tTimeout := DEFAULT_ADS_TIMEOUT);
	FrameStatisticClearCRC									:	FB_EcMasterFrameStatisticClearCRC:= (tTimeout := DEFAULT_ADS_TIMEOUT);
	FrameStatisticClearFrames								:	FB_EcMasterFrameStatisticClearFrames:= (tTimeout := DEFAULT_ADS_TIMEOUT);
	FrameStatisticClearTxRxErr								:	FB_EcMasterFrameStatisticClearTxRxErr:= (tTimeout := DEFAULT_ADS_TIMEOUT);
	IoDevreset												:	IOF_DeviceReset := (TMOUT := DEFAULT_ADS_TIMEOUT);
END_VAR

	(* Read or set (ReqState <> 0) EtherCAT Master State			*)
	(****************************************************************)

(* Process ******************************************************)
	rtExecute(CLK := Execute);

	CASE state OF
	(* Cyclic reading of state ***********************************)
	0:
		Busy 												:= FALSE;
                                        					
		IF rtExecute.Q THEN            					
			Busy 											:= TRUE;
			Done 											:= FALSE;
			Error											:= FALSE;
			ErrorID											:= 0;
			Errortext										:= '';
			DevResetDone									:= FALSE;
			CurrState										:= 0;
			ReqStateOK										:= FALSE;
			StateText										:= '';
			GetMasterState(bExecute := FALSE,sNetId	:= AmsNetId);
			SetMasterState(bExecute := FALSE,sNetId	:= AmsNetId );
			ReadMasterFrameStatistic(bExecute := FALSE,sNetId	:= AmsNetId );
			FrameStatisticClearCRC(bExecute := FALSE,sNetId	:= AmsNetId );
			FrameStatisticClearFrames(bExecute := FALSE,sNetId	:= AmsNetId );
			FrameStatisticClearTxRxErr(bExecute := FALSE,sNetId	:= AmsNetId );
			IoDevReset(RESET := FALSE);
			TON_TimeoutSetStatus(IN := FALSE);

			IF ReqState <> 0 
				AND (ReqState <> CurrState OR ReqState <> MemReqState)
			THEN
				SetMasterState( bExecute	:= TRUE, reqState	:= ReqState);
				MemReqState 								:= ReqState;
				state 										:= SEL(Options.7, 10, 11) ; //Start with reset device
			ELSE
				(* Start Read Status *)
				GetMasterState(bExecute	:= TRUE);
				state 										:= 1;
			END_IF
		ELSIF NOT Execute THEN
			Done 											:= FALSE;
			DevResetDone 									:= FALSE;
			Error											:= FALSE;
			ErrorID											:= 0;
			ErrorText										:= '';
		END_IF                      					

	(* Read state ******************************************)
	1:
		GetMasterState(bExecute := TRUE);
		IF NOT GetMasterState.bBusy
		THEN
			IF GetMasterState.bError THEN
				Busy										:= FALSE;
				Error										:= TRUE;
				ErrorId										:= GetMasterState.nErrId;
				ErrorText									:= CONCAT('FB_EcGetMasterState Id: ',UDINT_TO_STRING(ErrorId));
				state 										:= 0;
			ELSE                
				CurrState									:= GetMasterState.state;
				ReqStateOK									:= CurrState = ReqState OR ReqState = 0;
				StateText									:= F_ConvStateToString(CurrState);							
				state 										:= state + 1;
			END_IF
		END_IF
		
	(* read frame statistic ******************************************)
	2:
		ReadMasterFrameStatistic(bExecute := TRUE);
		IF NOT ReadMasterFrameStatistic.bBusy
		THEN
			IF ReadMasterFrameStatistic.bError THEN
				Busy										:= FALSE;
				Error										:= TRUE;
				ErrorId										:= ReadMasterFrameStatistic.nErrId;
				ErrorText									:= CONCAT('FB_EcMasterFrameStatistic Id: ',UDINT_TO_STRING(ErrorId));
				state 										:= 0;
			ELSE                
				LostFrames 									:= ReadMasterFrameStatistic.nLostFrames;
				FramesPerSecond 							:= ReadMasterFrameStatistic.fFramesPerSecond;
				LostQueuedFrames 							:= ReadMasterFrameStatistic.nLostQueuedFrames;
				QueuedFramesPerSecond 						:= ReadMasterFrameStatistic.fQueuedFramesPerSecond;		
				state 										:= 20;
			END_IF
		END_IF
		
	(* Set state *****************************************)
	10:
		TON_TimeoutSetStatus(IN := TRUE, PT := TIMEOUT_SET_STATE);
		SetMasterState(bExecute := TRUE);
		IF NOT SetMasterState.bBusy
		THEN
			IF SetMasterState.bError AND DevResetDone
			THEN
				Busy										:= FALSE;
				Error										:= TRUE;
				ErrorId										:= SetMasterState.nErrId;
				ErrorText									:= CONCAT('FB_EcSetMasterState Id: ',UDINT_TO_STRING(ErrorId));
				state 										:= 0;
			ELSIF SetMasterState.currState = MemReqState 
			THEN
				CurrState									:= SetMasterState.currState;
				ReqStateOK									:= CurrState = ReqState;
				StateText									:= F_ConvStateToString(CurrState);			
				state 										:= 2;
			ELSIF DevResetDone          					
			THEN     
				Busy										:= FALSE;                   					
				Error										:= TRUE;
				ErrorId										:= E_AdsErr.DEVICE_ABORTED;
				ErrorText									:= 'Device Reset failed - Master state <> ReqState';
				state 										:= 0;
			ELSE //Try to reset master 
				state 										:= state + 1;
			END_IF                      	
            SetMasterState(bExecute := FALSE);                            	
		ELSIF TON_TimeoutSetStatus.Q 
		THEN
			IF NOT DevResetDone 
			THEN (* try to reset master one time  *)
				state 										:= state + 1;
				IoDevReset(RESET := FALSE);
			ELSE
				Busy										:= FALSE;
				ErrCntReset 								:= ErrCntReset +1;
				Error										:= TRUE;
				ErrorId										:= E_AdsErr.DEVICE_TIMEOUT;
				ErrorText									:= CONCAT('FB_EcSetMasterState busy for more then ', TO_STRING(TIMEOUT_SET_STATE));
				state 										:= 0;
			END_IF  
			SetMasterState(bExecute := FALSE);                						
		END_IF

	11:
		TON_TimeoutSetStatus(IN := FALSE);
		state 												:= state + 1;

	(* Reset Device by setting Error State  **********************)
	12:	
		IoDevReset(DEVICEID	:= DevId,RESET	:= TRUE );
		IF NOT IoDevReset.BUSY
		THEN
			IF IoDevReset.ERR THEN
				Busy										:= FALSE;
				Error										:= TRUE;
				ErrorId										:= IoDevReset.ERRID;
				ErrorText									:= CONCAT('IOF_DeviceReset Id: ',UDINT_TO_STRING(ErrorId));
				state 										:= 0;
			ELSE //Tr to                         					
				Error										:= FALSE;
				ErrorId										:= 0;
				ErrorText									:= '';
				DevResetDone 								:= TRUE;
				TON_TimeoutSetStatus(IN := FALSE);
				state 										:= 10;
			END_IF
		ELSE
			;
		END_IF
		
	(* Start to clear frame statistic **********************************)
	20: 
		FrameStatisticClearCRC(bExecute := Options.0);
		IF NOT FrameStatisticClearCRC.bBusy
		THEN
			IF FrameStatisticClearCRC.bError THEN
				Busy										:= FALSE;
				Error										:= TRUE;
				ErrorId										:= FrameStatisticClearCRC.nErrId;
				ErrorText									:= CONCAT('FB_EcMasterFrameStatisticClearCRC Id: ',UDINT_TO_STRING(ErrorId));
				state 										:= 0;
			ELSE                
				state 										:= state + 1;
			END_IF
		END_IF		
	
	21: 
		FrameStatisticClearFrames(bExecute := Options.1);
		IF NOT FrameStatisticClearFrames.bBusy
		THEN
			IF FrameStatisticClearFrames.bError THEN
				Busy										:= FALSE;
				Error										:= TRUE;
				ErrorId										:= FrameStatisticClearFrames.nErrId;
				ErrorText									:= CONCAT('FB_EcMasterFrameStatisticClearFrames Id: ',UDINT_TO_STRING(ErrorId));
				state 										:= 0;
			ELSE                
				state 										:= state + 1;
			END_IF
		END_IF	

	22: 
		FrameStatisticClearTxRxErr(bExecute := Options.2);
		IF NOT FrameStatisticClearTxRxErr.bBusy
		THEN
			IF FrameStatisticClearTxRxErr.bError THEN
				Busy										:= FALSE;
				Error										:= TRUE;
				ErrorId										:= FrameStatisticClearTxRxErr.nErrId;
				ErrorText									:= CONCAT('FB_EcMasterFrameStatisticClearTxRxErr Id: ',UDINT_TO_STRING(ErrorId));
				state 										:= 0;
			ELSE                
				Busy										:= FALSE;
				Done										:= TRUE;
				state 										:= 0;
			END_IF
		END_IF	
		
	ELSE
		;
	END_CASE
                										
(*********************************************************************)

{attribute 'monitoring' := 'call'}
PROPERTY PUBLIC optClearCRCErrorCounter : BOOL
GET
optClearCRCErrorCounter := Options.0;
END_GET
SET
Options.0 := optClearCRCErrorCounter;
END_SET
END_PROPERTY

{attribute 'monitoring' := 'call'}
PROPERTY PUBLIC optClearLostFramesCounter : BOOL
GET
optClearLostFramesCounter := Options.1;
END_GET
SET
Options.1 := optClearLostFramesCounter;
END_SET
END_PROPERTY

{attribute 'monitoring' := 'call'}
PROPERTY PUBLIC optClearTCRXErrCounter : BOOL
GET
optClearTCRXErrCounter := Options.2;
END_GET
SET
Options.2 := optClearTCRXErrCounter;
END_SET
END_PROPERTY

{attribute 'monitoring' := 'call'}
PROPERTY PUBLIC optForceDevReset : BOOL
GET
optForceDevReset := Options.7;
END_GET
SET
Options.7 := optForceDevReset;
END_SET
END_PROPERTY

END_FUNCTION_BLOCK

// POUs/Fieldbus/EtherCAT/_Components/EcSlavesDiag
{attribute 'no_check'}
{attribute 'enable_dynamic_creation'}
FUNCTION_BLOCK EcSlavesDiag EXTENDS FbBase
VAR CONSTANT
	SLAVE_ADDR_OFFSET										:	UINT := 1000;
	DEL_SSTATE_CHANGED										:	 TIME := T#2S;
END_VAR
VAR_OUTPUT CONSTANT         								
	MIN_SLAVES												: 	UINT := 1;
	MAX_SLAVES												: 	UINT := PARAM.ETHERCAT_DIAG_MAX_SLAVES;	//EC_MAX_SLAVES = 65535 Slaves;
	
{attribute 'displaymode':='binary'}
	OPTION_READ_SCAN_SLAVES									:	BYTE := 2#0000_0001; //Read scanned slaves identity and link State
{attribute 'displaymode':='binary'}
	OPTION_SORT_INFO_DATA									:	BYTE := 2#0000_0010; //Sort list of slaves InfoData according to scanned/physical sequence
{attribute 'displaymode':='binary'}
	OPTION_UPDATE_TOPO_DATA									:	BYTE := 2#0000_0100; //Read topology data, helpful if hot connect groups are configured
{attribute 'displaymode':='binary'}
	OPTION_UPDATE_CONFIG_DATA								:	BYTE := 2#0000_1000; //Read info slave data with with every execution	
END_VAR           
VAR_INPUT
	MasterAmsNetId											:	T_AmsNetId;
{attribute 'displaymode':='binary'}
	Options													:	BYTE := 0;
END_VAR
VAR_OUTPUT         
	NoOfSlaves												:	UINT;			//shows number of configured slaves
	NoOfSlavesNOK											:	UINT;  			//Shows number of slaves not in OP or with CRC error etc
	NoOfHCGroups											:	UINT;  			//Shows number of hot connect groups
	NoOfHCSlaves											:	UINT;  			//Shows number of slave in a hot connect group
	InfoData												:	ARRAY [MIN_SLAVES..MAX_SLAVES] OF EC_SLAVE_DIAG_INFO_DATA; //configures slaves			
	LastActiveSlave											:	EC_SLAVE_DIAG_INFO_DATA;	//shows last slave in OP connected to port A 
	FirstErrorSlave											:	EC_SLAVE_DIAG_INFO_DATA;	//shows first slave with an error
	InfoDataSorted											:	BOOL; //Info data list sorted according physical sequence vs. configured seq.
	InvalidVPRS												:	BOOL; //Invalid VPRS active
	ErrorText												:	T_MAXSTRING;//shows error text of FB
	ExecutionTime											: 	TIME; //Total cycle time to execute the FB
END_VAR                     								         								
VAR                         								
(* Cache ********************************************************)               								
	pMemory													:	POINTER TO BYTE;
	SizeOfMemory											:	UDINT;
	MemNoOfSlaves											:	UINT;	
	ScannedSeqMixed											:	BOOL; //Scanned slave sequence is different to configured 

	pScannedSlaves											:	POINTER TO ARRAY [MIN_SLAVES..MAX_SLAVES] OF Tc2_EtherCAT.ST_EcSlaveScannedData;
	pConfigSlaves											:	POINTER TO ARRAY [MIN_SLAVES..MAX_SLAVES] OF Tc2_EtherCAT.ST_EcSlaveConfigData; 
	pSlavesState											:	POINTER TO ARRAY [MIN_SLAVES..MAX_SLAVES] OF Tc2_EtherCAT.ST_EcSlaveState;
	pSlavesStatusCode										:	POINTER TO ARRAY [MIN_SLAVES..MAX_SLAVES] OF DWORD;
	pTopologyData											:	POINTER TO ARRAY [MIN_SLAVES..MAX_SLAVES] OF Tc2_EtherCAT.ST_TopologyDataEx;
	
	StartTime												:	TIME;
	
(* timer ********************************************************)

(* trigger ********************************************************)

(* function-blocks *************************************************)
	EcGetSlaveCount											:	FB_EcGetSlaveCount := (tTimeout	:= T#60S);
	EcGetConfSlaves											:	FB_EcGetConfSlaves := (tTimeout	:= T#60S);
	EcGetScannedSlaves										:	FB_EcGetScannedSlaves := (tTimeout	:= T#60S);
	EcGetAllSlaveStateS										:	FB_EcGetAllSlaveStateS := (tTimeout	:= T#60S);
	EcGetAllSlaveCrcErrors									:	FB_EcGetAllSlaveCrcErrors := (tTimeout	:= T#60S);
	EcGetAllSlaveAbnormalStateChanges						:	FB_EcGetAllSlaveAbnormalStateChanges := (tTimeout	:= T#60S);	
	EcGetSlaveTopologyInfo									: 	FB_EcGetSlaveTopologyInfo := (tTimeout	:= T#60S);	
	
(* dummy **********************************************************)
	i,k,idx													:	UINT := 0;
	
END_VAR

	(* Check EtherCAT slaves status			V1	*)
	(********************************************)

(* Sequence *********************************)
	rtExecute(CLK := Execute);

	CASE State OF
	0:
		Busy 												:= FALSE;
		IF rtExecute.Q
		THEN //Clear data if FB is disabled or started
			Busy 											:= TRUE;
			Done											:= FALSE;
			Error											:= FALSE;
			Errorid											:= 0;
			ErrorText										:= '';	

		//	NoOfSlavesNIO									:= 0;	
			InvalidVPRS										:= FALSE;
			ScannedSeqMixed									:= FALSE;

			StartTime										:= TIME();
			ExecutionTime									:= T#0MS;
			
			EcGetSlaveCount(bExecute := FALSE,sNetId := MasterAmsNetId);
			EcGetConfSlaves(bExecute := FALSE,sNetId := MasterAmsNetId);
			EcGetSlaveTopologyInfo(bExecute := FALSE,sNetId := MasterAmsNetId);
			EcGetAllSlaveStates(bExecute := FALSE, sNetId := MasterAmsNetId);
			EcGetAllSlaveCrcErrors(bExecute := FALSE,sNetId := MasterAmsNetId);
			EcGetAllSlaveAbnormalStateChanges(bExecute := FALSE,sNetId := MasterAmsNetId);
			EcGetScannedSlaves(bExecute := FALSE,sNetId := MasterAmsNetId);
			
			MEMSET(ADR(LastActiveSlave),0,SIZEOF(LastActiveSlave));
			MEMSET(ADR(FirstErrorSlave),0,SIZEOF(FirstErrorSlave));
			
			IF NoOfSlaves = 0
			THEN
				State										:= 1;
			ELSIF Options.3 OR EcGetConfSlaves.nTotalSlaves = 0 OR InfoDataSorted
			THEN //Read config it not done or enabled
				State										:= 2;
			ELSIF Options.2 OR EcGetSlaveTopologyInfo.nSlaves = 0 OR InfoDataSorted
			THEN
				State										:= 10;
			ELSE
				State										:= 20;
			END_IF
		ELSIF NOT Execute
		THEN
			Done											:= FALSE;
			Error											:= FALSE;
			Errorid											:= 0;
			ErrorText										:= '';	
		END_IF
		IF StartTime > T#0MS AND ExecutionTime = T#0MS
		THEN
			ExecutionTime									:= TIME() - StartTime;
		END_IF
	
	(* Read no of found slaves *********************************************************************)
	1:
		EcGetSlaveCount(bExecute := NoOfSlaves = 0);
		IF NOT EcGetSlaveCount.bBusy
		THEN
			IF EcGetSlaveCount.bError 
			THEN
				Busy										:= FALSE;
				Error										:= TRUE;
				ErrorId										:= EcGetSlaveCount.nErrId;
				ErrorText									:= CONCAT('EcGetSlaveCount Id: ',UDINT_TO_STRING(ErrorId));
				State 										:= 0;
			ELSIF EcGetSlaveCount.nSlaves > MAX_SLAVES
			THEN			
				Busy										:= FALSE;
				Error										:= TRUE;
				ErrorId										:= E_AdsErr.DEVICE_INVALIDSIZE  ;
				ErrorText									:= CONCAT('No of slaves > PARAM.ETHERCAT_MASTER_DIAG_MAX_SLAVES, please update value to ', TO_STRING(EcGetSlaveCount.nSlaves));
				State										:= 0;  	
			ELSIF EcGetSlaveCount.bExecute AND NoOfSlaves <> EcGetSlaveCount.nSlaves
			THEN
				NoOfSlaves									:= EcGetSlaveCount.nSlaves;					

				//Init Info Data 	
				MEMSET(ADR(InfoData),0,SIZEOF(InfoData));

				k 											:= NoOfSlaves + 1;
				//Set buffer lenght according to needed memory space
				EcGetConfSlaves.cbBufLen					:= SIZEOF(Tc2_EtherCAT.ST_EcSlaveConfigData) * k;
				EcGetScannedSlaves.cbBufLen					:= SIZEOF(Tc2_EtherCAT.ST_EcSlaveScannedData) * k;
				EcGetAllSlaveStates.cbBufLen				:= SIZEOF(Tc2_EtherCAT.ST_EcSlaveState) * k;
				EcGetAllSlaveCrcErrors.cbBufLen				:= SIZEOF(DWORD) * k;	
				EcGetSlaveTopologyInfo.cbBufLen				:= SIZEOF(Tc2_EtherCAT.ST_TopologyDataEx) * k;	
				EcGetAllSlaveAbnormalStateChanges.cbBufLen	:= EcGetAllSlaveCrcErrors.cbBufLen;						
					
				//Allocate dynamic buffer memory 
				IF Allocate(MAX(EcGetSlaveTopologyInfo.cbBufLen,MAX(MAX(EcGetConfSlaves.cbBufLen,EcGetAllSlaveCrcErrors.cbBufLen), MAX(EcGetScannedSlaves.cbBufLen,EcGetAllSlaveStateS.cbBufLen) )))
				THEN
					//Write buffer lenght per FB	
					pConfigSlaves							:= pMemory;
					pScannedSlaves							:= pMemory;
					pSlavesState							:= pMemory;
					pSlavesStatusCode						:= pMemory;	
					pTopologyData							:= pMemory;	
					
					State 									:= State + 1;			
				ELSE
					Busy									:= FALSE;
					Error									:= TRUE;
					ErrorId									:= E_AdsErr.DEVICE_NOMEMORY; //No memory
					ErrorText								:= CONCAT('EcSlavesDiag.allocate() Id: ',UDINT_TO_STRING(ErrorId));
					NoOfSlaves								:= 0;
					State 									:= 0;	
				END_IF

			ELSE
				State 										:= State + 1;
			END_IF
		ELSE
			;
		END_IF		
	
	
	(* Read slaves "configuration" ************************************************************************************************************)
	2:
		EcGetConfSlaves(bExecute := TRUE, pArrEcConfSlaveInfo := pConfigSlaves, cbBufLen := (* See State 1 *) );
			
		IF NOT EcGetConfSlaves.bBusy
		THEN
			IF EcGetConfSlaves.bError 
			THEN
				Busy										:= FALSE;
				Error										:= TRUE;
				ErrorId										:= EcGetConfSlaves.nErrorId;
				ErrorText									:= CONCAT('FB_EcGetConfSlaves Id: ',UDINT_TO_STRING(ErrorId));
				State										:= 0;     
					
			ELSIF EcGetConfSlaves.nSlaves > MAX_SLAVES
			THEN
				Busy										:= FALSE;
				Error										:= TRUE;
				ErrorId										:= E_AdsErr.DEVICE_INVALIDSIZE  ;
				ErrorText									:= CONCAT('No of config slaves > PARAM.ETHERCAT_MASTER_DIAG_MAX_SLAVES, please update value to ', TO_STRING(EcGetConfSlaves.nSlaves));
				State										:= 0;  					
			ELSE
				State 										:= State + 1;
			END_IF
		END_IF	
			
	3: //Fill structure	
		k													:= MIN(EcGetConfSlaves.nSlaves, NoOfSlaves);
		FOR i := MIN_SLAVES TO k DO
			InfoData[i].Addr								:= pConfigSlaves^[i].nAddr;
			InfoData[i].ConfigType							:= pConfigSlaves^[i].sType; 
		//	InfoData[i].DevType								:= pConfigSlaves^[i].nDevType;
			InfoData[i].ConfigName							:= DELETE(pConfigSlaves^[i].sName, LEN(InfoData[i].ConfigType) + 3 , FIND(pConfigSlaves^[i].sName,InfoData[i].ConfigType) - 1); //Delete type if in brakets 	
			InfoData[i].ConfigTypeIdentity					:= F_ConvProductCodeToString(pConfigSlaves^[i].stSlaveIdentity);
			InfoData[i].ConfigIdentity						:= pConfigSlaves^[i].stSlaveIdentity;
		//	InfoData[i].LinkState							:= pConfigSlaves^[i].nLinkStatus; see read slaves state					
		END_FOR
		
		State 												:= SEL(Options.2 OR EcGetSlaveTopologyInfo.nSlaves = 0 OR InfoDataSorted, 20, 10);	
		
	(* Read slaves "topology" information *******************************************************************************************************)
	10:
		EcGetSlaveTopologyInfo(bExecute := NoOfSlaves > 0 , sNetId	:= MasterAmsNetId,  pAddrBuf := pTopologyData,  cbBufLen	:= (* See State 1 *));
		IF NOT EcGetSlaveTopologyInfo.bBusy
		THEN
			IF EcGetSlaveTopologyInfo.bError 
			THEN
				Busy										:= FALSE;
				Error										:= TRUE;
				ErrorId										:= EcGetSlaveTopologyInfo.nErrId;
				ErrorText									:= CONCAT('EcGetSlaveTopologyInfo Id: ',UDINT_TO_STRING(ErrorId));
				State 										:= 0;
			ELSIF EcGetSlaveTopologyInfo.nSlaves > MAX_SLAVES
			THEN
				Busy										:= FALSE;
				Error										:= TRUE;
				ErrorId										:= E_AdsErr.DEVICE_INVALIDSIZE  ;
				ErrorText									:= CONCAT('No of scanned slaves > PARAM.ETHERCAT_MASTER_DIAG_MAX_SLAVES, please update value to ', TO_STRING(EcGetScannedSlaves.nSlaves));
				State										:= 0;  	
			ELSE
				State 										:= State + 1;
			END_IF
		ELSE
			;
		END_IF	

	11:	//Fill structure		
		NoOfHCGroups										:= 0;
		NoOfHCSlaves										:= 0;
		k													:= MIN(EcGetSlaveTopologyInfo.nSlaves, NoOfSlaves);
		FOR i := MIN_SLAVES TO k DO                 		
			InfoData[i].TopoOwnPhysicalAddr					:= pTopologyData^[i].nOwnPhysicalAddr; 
			InfoData[i].TopologyStatus						:= pTopologyData^[i].nStatusBits;
			InfoData[i].HCSlaveCountCfg  					:= pTopologyData^[i].nHCSlaveCountCfg;
			InfoData[i].HCSlaveCountAct  					:= pTopologyData^[i].nHCSlaveCountAct;
			InfoData[i].AutoIncAddr   						:= pTopologyData^[i].nOwnAutoIncAddr;
			InfoData[i].PhysicalPortAddr    				:= pTopologyData^[i].stPhysicalAddr;
			InfoData[i].AutoIncPortAddr    					:= pTopologyData^[i].stAutoIncAddr;
			                                        		
			InfoData[i].HotConnectNodeStart 				:= InfoData[i].TopologyStatus.3;
			InfoData[i].HotConnectSlave 					:= InfoData[i].TopologyStatus.4;
                                                    		
			NoOfHCGroups									:= SEL(InfoData[i].HotConnectNodeStart , NoOfHCGroups, NoOfHCGroups + 1);
			NoOfHCSlaves									:= SEL(InfoData[i].HotConnectSlave , NoOfHCSlaves, NoOfHCSlaves + 1);
			                                        	
		END_FOR				                        	
		State 												:= 20;
		
	(* Read slaves "EtherCAT State and link state" ***************************************************************************************)
	20	:
		EcGetAllSlaveStateS(bExecute := NoOfSlaves > 0, pStateBuf:=  pSlavesState, cbBufLen	:= (* See State 1 *));
					
		IF NOT EcGetAllSlaveStateS.bBusy
		THEN
			IF EcGetAllSlaveStateS.bError 
			THEN
				Busy										:= FALSE;
				Error										:= TRUE;
				ErrorId										:= EcGetAllSlaveStateS.nErrId;
				ErrorText									:= CONCAT('FB_EcGetAllSlaveStates Id: ',UDINT_TO_STRING(ErrorId));
				State 										:= 0;
			ELSE
				k											:= MIN(EcGetAllSlaveStateS.nSlaves, NoOfSlaves);
				FOR i := MIN_SLAVES TO k DO
					InfoData[i].LinkState					:= pSlavesState^[i].linkState;
					InfoData[i].DevState					:= pSlavesState^[i].deviceState;
					InfoData[i].DevStateText				:= F_ConvSlaveStateToString(pSlavesState^[i]);
					InfoData[i].DevStateBits				:= F_ConvSlaveStateToBitsEx(pSlavesState^[i]);	
					InfoData[i].ErrorIdentCode.0			:= InfoData[i].DevStateBits.bInvVPRS; //Wrong slave
					IF InfoData[i].ErrorIdentCode.0 THEN InvalidVPRS := TRUE; END_IF
					InfoData[i].ErrorIdentCode.1			:= NOT InfoData[i].ErrorIdentCode.0 AND NOT InfoData[i].DevStateBits.bOp AND_THEN(NOT InfoData[i].HotConnectSlave OR NOT InfoData[i].DevStateBits.bInit); //Wrong State
				END_FOR	

				State 										:= State + 1;
			END_IF
		ELSE
			;
		END_IF	
		
	(* Get all slaves "CRC counter" ********************************************************************)
	21:	
		EcGetAllSlaveCrcErrors(bExecute := NoOfSlaves > 0, sNetId	:= MasterAmsNetId,  pCrcErrorBuf:= pSlavesStatusCode,  cbBufLen	:= (* See State 1 *));
		IF NOT EcGetAllSlaveCrcErrors.bBusy
		THEN
			IF EcGetAllSlaveCrcErrors.bError 
			THEN
				Busy										:= FALSE;
				Error										:= TRUE;
				ErrorId										:= EcGetAllSlaveStateS.nErrId;
				ErrorText									:= CONCAT('FB_EcGetAllSlaveCrcErrors Id: ',UDINT_TO_STRING(ErrorId));
				State 										:= 0;
			ELSE
				k											:= MIN(EcGetAllSlaveCrcErrors.nSlaves, NoOfSlaves);
				FOR i := MIN_SLAVES TO k DO
					InfoData[i].ErrorIdentCode.2			:= InfoData[i].CntOfCRCErrors <> pSlavesStatusCode^[i] AND pSlavesStatusCode^[i] > 0; //CRC error increased
					InfoData[i].CntOfCRCErrors				:= pSlavesStatusCode^[i];				
				END_FOR				
				
				State 										:= State + 1;
			END_IF
		ELSE
			;
		END_IF
		
	(* Get all slaves "no of abnormal state change" *****************************************************************************)
	22:	
		EcGetAllSlaveAbnormalStateChanges(bExecute := NoOfSlaves > 0, sNetId	:= MasterAmsNetId,  pAddrBuf := pSlavesStatusCode,  cbBufLen	:= (* See State 1 *));
		IF NOT EcGetAllSlaveAbnormalStateChanges.bBusy
		THEN
			IF EcGetAllSlaveAbnormalStateChanges.bError 
			THEN
				Busy										:= FALSE;
				Error										:= TRUE;
				ErrorId										:= EcGetAllSlaveAbnormalStateChanges.nErrId;
				ErrorText									:= CONCAT('FB_EcGetAllSlaveAbnormalStateChanges Id: ',UDINT_TO_STRING(ErrorId));
				State 										:= 0;
			ELSE
				k											:= MIN(EcGetAllSlaveAbnormalStateChanges.nSlaves, NoOfSlaves);
				FOR i := MIN_SLAVES TO k DO
					InfoData[i].ErrorIdentCode.3			:= InfoData[i].NoOfAbnormalStateChanges <> pSlavesStatusCode^[i] AND pSlavesStatusCode^[i] > 0; //Abnormal State change increased
					InfoData[i].NoOfAbnormalStateChanges	:= pSlavesStatusCode^[i];	
				END_FOR				
				
				State 										:= SEL(Options.0 OR EcGetScannedSlaves.nSlaves = 0, 40, 30);
			END_IF
		ELSE
			;
		END_IF

	(* Start to read scanned slaves *************************************************************************)
	30:
		EcGetScannedSlaves(bExecute := TRUE, pArrEcScannedSlaveInfo  := pScannedSlaves, cbBufLen := (* See State 1 *));
			
		IF NOT EcGetScannedSlaves.bBusy
		THEN
			IF EcGetScannedSlaves.bError 
				AND EcGetScannedSlaves.nErrorId <> 1817 //device has a timeout -> not error if no slave is connected 
			THEN
				Busy										:= FALSE;
				Error										:= TRUE;
				ErrorId										:= EcGetScannedSlaves.nErrorId;
				ErrorText									:= CONCAT('FB_EcGetScannedSlaves Id: ',UDINT_TO_STRING(ErrorId));
				State										:= 0;     

			ELSIF EcGetScannedSlaves.nSlaves > MAX_SLAVES
			THEN
				Busy										:= FALSE;
				Error										:= TRUE;
				ErrorId										:= E_AdsErr.DEVICE_INVALIDSIZE  ;
				ErrorText									:= CONCAT('No of scanned slaves > PARAM.ETHERCAT_MASTER_DIAG_MAX_SLAVES, please update value to ', TO_STRING(EcGetScannedSlaves.nSlaves));
				State										:= 0;  			
			
			ELSE	
				FOR i := MIN_SLAVES TO NoOfSlaves 
				DO					
					InfoData[i].ScannedTypeIdentity			:= '<not present>';
					MEMSET(ADR(InfoData[i].ScannedIdentity),0,SIZEOF(InfoData[i].ScannedIdentity));								
					InfoData[i].DataLinkStatusReg			:= 0;	
					InfoData[i].ScannedSeq					:= 0;						
				END_FOR
				State 										:= SEL(EcGetScannedSlaves.nSlaves = 0, State + 1, 40);
			END_IF
		END_IF
		
	31: //Fill structure
		k													:= MIN(EcGetScannedSlaves.nSlaves,NoOfSlaves); //No of scanned slaves
		idx													:= 0;
		ScannedSeqMixed										:= FALSE;
		FOR i := MIN_SLAVES TO NoOfSlaves DO		
			IF i <= EcGetScannedSlaves.nSlaves
			THEN
				idx											:= SEL(pScannedSlaves^[i].nAddr > SLAVE_ADDR_OFFSET, idx + 1 ,pScannedSlaves^[i].nAddr - SLAVE_ADDR_OFFSET);
				InfoData[idx].ScannedTypeIdentity			:= F_ConvProductCodeToString(pScannedSlaves^[i].stSlaveIdentity);
				InfoData[idx].ScannedIdentity				:= pScannedSlaves^[i].stSlaveIdentity;				
				InfoData[idx].DataLinkStatusReg				:= pScannedSlaves^[i].ndlStatusReg;		
				InfoData[idx].ScannedSeq					:= i;	
				ScannedSeqMixed								:= i <> idx OR ScannedSeqMixed;
			ELSE
				EXIT;
			END_IF
		
		END_FOR
		
		State 												:= 40;
		
	(* Search for error slaves **************************************************************************)
	40:
		k													:= EcGetScannedSlaves.nSlaves + 1; 
		NoOfSlavesNOK										:= 0;
		FOR i := MIN_SLAVES TO NoOfSlaves				
		DO
			//Fill PhysicalSeq number of missed slaves for possible sorting
			IF ScannedSeqMixed AND Options.1
			THEN
				IF InfoData[i].ScannedSeq = 0
				THEN 										
					InfoData[i].ScannedSeq 					:= k;
					k										:= k + 1;
				END_IF
			END_IF
		
			//Search for first slave with error
			IF InfoData[i].ErrorIdentCode <> 0
			THEN
				NoOfSlavesNOK								:= NoOfSlavesNOK + 1;
				IF FirstErrorSlave.Addr = 0
				THEN
					FirstErrorSlave 						:= InfoData[i]; 					
					IF i - 1 > 0
					THEN
						LastActiveSlave 					:= InfoData[i - 1];
					END_IF
				END_IF						
			END_IF
		END_FOR   	
	
		IF ScannedSeqMixed AND Options.1
		THEN
			InfoDataSorted									:= TRUE;
			State											:= State + 1;
		ELSE
			InfoDataSorted									:= FALSE;
			Busy											:= FALSE;
			Done											:= TRUE;
			State											:= 0;   
		END_IF
	
	(* Sort InfoData list if sequence is mixed and option selected **************************************************************************)	
	41: 
		IF sortList()
		THEN
			Busy											:= FALSE;
			Done											:= TRUE;
			State											:= 0;   
		ELSE
			Busy											:= FALSE;
			Error											:= TRUE;
			ErrorId											:= E_AdsErr.DEVICE_INVALIDDATA  ; //Invalid data
			ErrorText										:= 'Error sorting InfoData list ';
			State											:= 0;  			
		END_IF	
 
	ELSE
		;
	END_CASE

(***********************************************************************)

METHOD PROTECTED FINAL allocate : BOOL
VAR_INPUT 
	MemSize													:	UDINT;
END_VAR
VAR
END_VAR
IF MemSize = 0
THEN
	allocate												:= FALSE;	
ELSIF pMemory = 0 
THEN
	pMemory													:= __NEW(BYTE,MemSize );
	SizeOfMemory											:= MemSize;
	IF PARAM.ENABLE_DEBUG_MSG_DYNAMIC_MEM_ALLOCATION
	THEN
		AdsLogHint('EngineeringToolbox | FB EcSlavesDiag | An instance allocated %s bytes from the dynamic memory of the ADS router memory pool', TO_STRING(MemSize));
	END_IF
	Allocate												:= TRUE;	
ELSIF MemSize > SizeOfMemory
THEN//Size increased, allocate new memory
	__DELETE(pMemory);  //Delete reference to old memory
	
	pMemory													:= __NEW(BYTE,MemSize );
	SizeOfMemory											:= MemSize;
	IF PARAM.ENABLE_DEBUG_MSG_DYNAMIC_MEM_ALLOCATION
	THEN
		AdsLogWarn('EngineeringToolbox | FB EcSlavesDiag | No of slaves increased and one instance allocated additional %s bytes from the dynamic memory of the ADS router memory pool', TO_STRING(MemSize));
	END_IF

	Allocate												:= TRUE;
ELSE
	Allocate												:= FALSE;
END_IF
END_METHOD

METHOD FB_exit : BOOL
VAR_INPUT
	bInCopyCode : BOOL; // if TRUE, the exit method is called for exiting an instance that is copied afterwards (online change).
END_VAR
IF NOT bInCopyCode AND pMemory <> 0
THEN //Release memory in case the PLC stopps
	__DELETE(pMemory);
	SizeOfMemory								:= 0;
END_IF
END_METHOD

{attribute 'monitoring' := 'call'}
PROPERTY PUBLIC optReadScannedSlaves : bool
GET
optReadScannedSlaves := Options.0;
END_GET
SET
OPtions.0 := optReadScannedSlaves;
END_SET
END_PROPERTY

{attribute 'monitoring' := 'call'}
PROPERTY PUBLIC optSortInfoData : bool
GET
optSortInfoData := Options.2;
END_GET
SET
OPtions.2 := optSortInfoData;
END_SET
END_PROPERTY

{attribute 'monitoring' := 'call'}
PROPERTY PUBLIC optUpdateConfigData : bool
GET
optUpdateConfigData := Options.3;
END_GET
SET
OPtions.3 := optUpdateConfigData;
END_SET
END_PROPERTY

{attribute 'monitoring' := 'call'}
PROPERTY PUBLIC optUpdateTopoData : bool
GET
optReadScannedSlaves := Options.1;
END_GET
SET
OPtions.1 := optReadScannedSlaves;
END_SET
END_PROPERTY

METHOD INTERNAL sortList : BOOL
VAR_INPUT
END_VAR
VAR
	SlaveInfoData1											:	EC_SLAVE_DIAG_INFO_DATA;
	SlaveInfoData2											:	EC_SLAVE_DIAG_INFO_DATA;
END_VAR
	sortList												:= TRUE;
	
	i														:= MIN_SLAVES;
	WHILE i <= NoOfSlaves OR SlaveInfoData1.ScannedSeq <> 0 
	DO
		IF SlaveInfoData1.ScannedSeq > 0
		THEN
			IF SlaveInfoData1.ScannedSeq > NoOfSlaves
			THEN //Error seq no
				sortList									:= FALSE;
				EXIT;
			ELSE
				SlaveInfoData2 								:= InfoData[SlaveInfoData1.ScannedSeq]; //Backup target
				InfoData[SlaveInfoData1.ScannedSeq].ScannedSeq	:= 0; //Mark as copied				
				InfoData[SlaveInfoData1.ScannedSeq]			:= SlaveInfoData1; //Copy from cache into target	
				SlaveInfoData1								:= SlaveInfoData2; //Write backed up data into cache
			END_IF

		ELSIF InfoData[i].ScannedSeq > 0 AND InfoData[i].ScannedSeq <> i
		THEN
			//Put target into cache
			SlaveInfoData1									:= InfoData[InfoData[i].ScannedSeq];
			InfoData[InfoData[i].ScannedSeq]				:= InfoData[i];		
			InfoData[i].ScannedSeq							:= 0; //Mark as copied
		ELSE
			;				
		END_IF   
		i													:= i + 1;
	END_WHILE;
END_METHOD

END_FUNCTION_BLOCK

// POUs/Fieldbus/EtherCAT/_Components/EcSlaveSupervisor
{attribute 'no_check'}
(* Set EtherCAT state(ReqState <> 0) or read state and CRC error counter of EtherCAT slave *)
FUNCTION_BLOCK EcSlaveSupervisor Extends FbBase
VAR_INPUT
	EcMasterAmsNetId										:	T_AmsNetId;
	SlaveAddr												: 	UINT; 		//-> Slave Port number!
{attribute 'displaymode':='hex'}
	ReqState												:	WORD := 0; (* 	EC_DEVICE_STATE_INIT		:BYTE 	:=16#01;
																				EC_DEVICE_STATE_PREOP		:BYTE 	:=16#02;
																				EC_DEVICE_STATE_BOOTSTRAP	:BYTE 	:=16#03;
																				EC_DEVICE_STATE_SAFEOP		:BYTE 	:=16#04;
																				EC_DEVICE_STATE_OP			:BYTE 	:=16#08; *)																				
END_VAR                     							
VAR_OUTPUT                  							
{attribute 'displaymode':='hex'}
	CurrState												: 	BYTE;	(* Shows current state 																					
																				EC_DEVICE_STATE_INIT		:BYTE 	:=16#01;
																				EC_DEVICE_STATE_PREOP		:BYTE 	:=16#02;
																				EC_DEVICE_STATE_BOOTSTRAP	:BYTE 	:=16#03;
																				EC_DEVICE_STATE_SAFEOP		:BYTE 	:=16#04;
																				EC_DEVICE_STATE_OP			:BYTE 	:=16#08; *)
{attribute 'displaymode':='hex'}
	linkState												: 	BYTE;	(* Shows state of link
																				EC_LINK_STATE_OK :BYTE :=16#00;
																				EC_LINK_STATE_NOT_PRESENT :BYTE :=16#01;
																				EC_LINK_STATE_LINK_WITHOUT_COMM :BYTE :=16#02;
																				EC_LINK_STATE_MISSING_LINK :BYTE :=16#04;
																				EC_LINK_STATE_ADDITIONAL_LINK :BYTE :=16#08;
																				EC_LINK_STATE_PORT_A :BYTE :=16#10;
																				EC_LINK_STATE_PORT_B :BYTE :=16#20;
																				EC_LINK_STATE_PORT_C :BYTE :=16#40;
																				EC_LINK_STATE_PORT_D :BYTE :=16#80; *)
																				
	ReqStateOK												:	BOOL;		//Requested state of slave is OK
	StateBits												:	ST_EcSlaveStateBitsEx;
	StateText												:	STRING(80);	//State as text
	CrcError    											:    ST_EcCrcErrorEx; (*Crc error of the EtherCAT slave device*)
END_VAR                 								
VAR                     								
	TON_GetStateTrig										:	TON;
	SetSlaveState											:	FB_EcSetSlaveSTATE := (tTimeout := DEFAULT_ADS_TIMEOUT);
	GetSlaveState											:	FB_EcGetSlaveSTATE := (tTimeout := DEFAULT_ADS_TIMEOUT);
	GetSlaveCrcErrorEx 										:	FB_EcGetSlaveCrcErrorEx  := (tTimeout := DEFAULT_ADS_TIMEOUT);
	MemReqState												:	WORD;
	ErrorText												:	STRING(40);
END_VAR

	(* Set EtherCAT state(ReqState <> 0) or read state and CRC error counter of EtherCAT slave *)
	(*******************************************************************************************)

(* Process ******************************************************)
	rtExecute(CLK := Execute);

	CASE state OF
	(* cyclic reading of state ***********************************)
	0:
		Busy 												:= FALSE;

		IF rtExecute.Q 
		THEN
			Busy 											:= TRUE;
			Done											:= FALSE;
			Error											:= FALSE;
			ErrorID											:= 0;
			Errortext										:= '';
			CurrState										:= 0;
			linkState										:= 0;
			ReqStateOK										:= FALSE;
			MEMSET(ADR(StateBits),0,SIZEOF(StateBits));
			MEMSET(ADR(CrcError),0,SIZEOF(CrcError));	
			StateText										:= '';
	
			SetSlaveSTATE(bExecute := FALSE, sNetId:= EcMasterAmsNetId,nSlaveAddr:= SlaveAddr);
			GetSlaveSTATE(bExecute := FALSE,sNetId:= EcMasterAmsNetId,nSlaveAddr:= SlaveAddr);
			GetSlaveCrcErrorEx(bExecute := FALSE,sNetId:= EcMasterAmsNetId,nSlaveAddr:= SlaveAddr);

			IF(ReqState <> CurrState
				OR ReqState <> MemReqState)
				AND ReqState <> 0
			THEN
				SetSlaveState(bExecute:= TRUE,reqState:= ReqState);
				MemReqState 								:= ReqState;
				state 										:= 10;

			ELSE
				(* Start Reading State *)
				GetSlaveState(bExecute	:= TRUE);
				state 										:= 1;
			END_IF

		ELSIF NOT Execute 
		THEN
			Done 											:= FALSE;
			Error											:= FALSE;
			ErrorID											:= 0;
			ErrorText										:= '';
		END_IF

	(* Read Slave State **************************************)
	1:
		(* Work block *)
		GetSlaveState();

		IF NOT GetSlaveState.bBusy
		THEN
			IF GetSlaveState.bError THEN
				Busy										:= FALSE;
				Error										:= TRUE;
				ErrorId										:= GetSlaveState.nErrId;
				ErrorText									:= CONCAT('FB_EcGetSlaveSTATE Id: ',UDINT_TO_STRING(ErrorId));
				state 										:= 0;
			ELSE       
				ReqStateOK 									:= (ReqState = CurrState OR ReqState = 0);         					
				CurrState 									:= GetSlaveState.state.deviceState;
				linkState 									:= GetSlaveState.State.linkState;
				StateText 									:= F_ConvStateToString(GetSlaveState.State.deviceState);
			 	StateBits							 		:= F_ConvSlaveStateToBitsEx(GetSlaveState.state);
				state										:= state + 1;
			END_IF
			GetSlaveSTATE(bExecute := FALSE);
		ELSE
			;
		END_IF

	(* Read Slave CRC Error Counter  **************************************)		
	2: 
		(* Work block *)
		GetSlaveCrcErrorEx();

		IF NOT GetSlaveCrcErrorEx.bBusy
		THEN
			IF GetSlaveCrcErrorEx.bError THEN
				Busy										:= FALSE;
				Error										:= TRUE;
				ErrorId										:= GetSlaveCrcErrorEx.nErrId;
				ErrorText									:= CONCAT('FB_EcGetSlaveCrcErrorEx Id: ',UDINT_TO_STRING(ErrorId));
				state 										:= 0;
			ELSE       
				CrcError									:= 	GetSlaveCrcErrorEx.crcError;
				Done 										:= TRUE;
				Busy 										:= FALSE;
				state										:= 0;
			END_IF
			GetSlaveCrcErrorEx(bExecute := FALSE);
		ELSE
			;
		END_IF

	(* Set state  *****************************************)
	10:	
		SetSlaveState();  
		IF NOT SetSlaveState.bBusy
		THEN
			IF SetSlaveState.bError 
			THEN             	
				Busy										:= FALSE;
				Error										:= TRUE;
				ErrorId										:= SetSlaveState.nErrId;
				ErrorText									:= CONCAT('FB_EcSetSlaveSTATE Id: ',UDINT_TO_STRING(ErrorId));
				state 										:= 0;
			ELSIF SetSlaveState.CurrState.deviceState = MemReqState 
			THEN
				ReqStateOK									:= TRUE;
				Busy 										:= FALSE;
				Done 										:= TRUE;	
				state 										:= 0;
			ELSE                    				
				Busy										:= FALSE;		
				Error										:= TRUE;
				ErrorId										:= E_AdsErr.DEVICE_ABORTED;
				ErrorText									:= 'SetSlaveState DEVICESTATE <> ReqState';
				state	 									:= 0;
			END_IF         					
			CurrState 										:= SetSlaveState.currState.deviceState;
			linkState 										:= SetSlaveState.currState.linkState;
			StateText 										:= F_ConvStateToString(SetSlaveState.currState.deviceState);
			StateBits							 			:= F_ConvSlaveStateToBitsEx(SetSlaveState.currState);
			SetSlaveState(bExecute := FALSE);              						
		END_IF                      						
	END_CASE


(*********************************************************************)

END_FUNCTION_BLOCK

// POUs/Fieldbus/EtherCAT/EcCoEReadNewestDiagMsg
{attribute 'no_check'}
//Read EtherCAT diag newest message from EtherCAT slave via CoE
FUNCTION_BLOCK EcCoEReadNewestDiagMsg EXTENDS fbBase      
VAR CONSTANT
	{attribute 'displaymode':='hexadecimal'} 
	COE_DIAG_OBJECT											: WORD := 16#10F3;
END_VAR                  						
VAR_INPUT                           						
	AdsAddr													: 	AMSADDR; //Terminal AMS Net Addr.
	Timeout													:	TIME := DEFAULT_ADS_TIMEOUT;
END_VAR
VAR_IN_OUT
END_VAR
VAR_OUTPUT
	{attribute 'displaymode':='hexadecimal'}
	Message													: ARRAY[0..63] OF BYTE; //Index A010 with a lenght of 27 or 32/64 bytes subindex
	{attribute 'displaymode':='hexadecimal'}
	DiagCode												: UDINT; // first 4 bytes of message

	{attribute 'displaymode':='hexadecimal'}
	TextId													: UINT; //xyzz -> X =Type | y = Source | zz = Message ID
	Timestamp												: T_DCTIME64;	

	MsgSeverity												: UINT; //Extracted from Flags ->  -> 0:Info | 1:Warning | 2:Error 
	MsgTimestampLocal										: BOOL; //Extracted from Flags bit 4
	MsgNoOfParameter										: UINT; //Extracted from Flags 

	{attribute 'displaymode':='hexadecimal'}
	MsgType													: UINT; //Extracted from TextId -> 0=SystemInfo | 1:Info | 2:reserved | 4:Warning | 8:Error
	MsgSource												: UINT; //Extracted from TextId -> 0:System | 1:General | 2:Communication | 3:Encoder | 4:Drive | 5:Inputs | 6:IO | 7:Reserved 
	{attribute 'displaymode':='hexadecimal'}
	MsgId													: UINT; //Extracted from TextId 
END_VAR                             						
VAR

END_VAR
VAR
(* Cache *********************************************************************)	
	{attribute 'displaymode':='hexadecimal'}
	SubIndexNewestMessage									: BYTE;

	{attribute 'displaymode':='hexadecimal'}
	Flags													: UINT; //Info (0) Warning (1) or Error (2)
(* Timer ********************************************************************************)
  	
(* Trigger ******************************************************************************)


(* Function blocks ****************************************************************************)
	CoERead													: FB_EcCoeSdoReadEx;

(* Dummy Speicher **********************************************************)
	
END_VAR

	(* Read newest diag message															*)
	(************************************************************************************)

(* Sequence *****************************************************************)
	rtExecute(CLK := Execute);
	CASE state OF
	0: // Read subindex of the newest diagnosis message		
		busy												:= FALSE;
		IF rtExecute.Q
		THEN
			Busy											:= TRUE;
			Done											:= FALSE;
			Error											:= FALSE;
			ErrorId											:= 0;
			CoERead(bExecute := FALSE, sNetId := F_CreateAmsNetId(nIds := AdsAddr.netId),  nSlaveAddr := AdsAddr.port, bCompleteAccess:= FALSE ,nIndex := COE_DIAG_OBJECT , tTimeout := Timeout);
			
			MEMSET(ADR(Message),0,SIZEOF(Message));
			DiagCode										:= 0;
			Flags											:= 0;
			TextId											:= 0;
			Timestamp										:= 0;
			MsgType											:= 0;
			MsgSource										:= 0;
			MsgId											:= 0;
			
			state											:= state + 1;
		ELSIF NOT Execute
		THEN
			Done											:= FALSE;
			Error											:= FALSE;
			ErrorId											:= 0;
		END_IF
	1: // read subindex of newest diagnosis message
		CoERead(
			bExecute	:= TRUE, //Diagnosis histroy object
			nSubIndex	:= 16#02, // subindex newest message
			pDstBuf		:= ADR(SubIndexNewestMessage), 
			cbBufLen	:= SIZEOF(SubIndexNewestMessage) );
				
		IF NOT CoERead.bBusy
		THEN
			IF CoERead.bError
			THEN
				Busy										:= FALSE;
				Error										:= TRUE;
				ErrorId										:= CoERead.nErrId;
				state										:= 0;
			ELSE		
				state										:= state + 1;
			END_IF			
			CoERead(bExecute := FALSE );				
		END_IF
		
	2: // Read newest diagnosis messages from sub index
		CoERead(
			bExecute	:= TRUE, 
			nSubIndex	:= SubIndexNewestMessage, 
			pDstBuf		:= ADR(Message), 
			cbBufLen	:= SIZEOF(Message));
			
		IF NOT CoERead.bBusy
		THEN
			IF CoERead.bError
			THEN
				Busy										:= FALSE;
				Error										:= TRUE;
				ErrorId										:= CoERead.nErrId;
				state										:= 0;				
			ELSE // Copy certain byte arrays of the diagnosis messages to lcoal variables
				
				MEMCPY(ADR(DiagCode), ADR(Message[0]), 4); 		// copy 4 bytes of diag code data
				MEMCPY(ADR(Flags), ADR(Message[4]), 2); 		// copy 2 bytes of flag data
				MEMCPY(ADR(TextID),ADR(Message[6]), 2);			// copy 2 bytes of TextId data
				MEMCPY(ADR(Timestamp),ADR(Message[8]), 8);		// copy 8 bytes of 64bit DC time
				
				MsgType										:= SHR(TextId AND 16#F000, 12);
				MsgSource									:= SHR(TextId AND 16#0F00, 8);
				MsgId										:= TextId AND 16#00FF;
				MsgSeverity									:= Message[4] AND 2#0000_1111;
				MsgTimestampLocal							:= Message[4].4;
				MsgNoOfParameter							:= Message[5];
				
				Done										:= TRUE;
				state										:= 0;			
			END_IF
			CoERead(bExecute := False);		
		END_IF
	END_CASE


(******************************************************************************)

{attribute 'monitoring' := 'call'}
PROPERTY PUBLIC msgSevyIsError : BOOL
GET
msgSevyIsError := MsgSeverity = 2;
END_GET
END_PROPERTY

{attribute 'monitoring' := 'call'}
PROPERTY PUBLIC msgSevyIsInfo : BOOL
GET
msgSevyIsInfo := MsgSeverity = 0;
END_GET
END_PROPERTY

{attribute 'monitoring' := 'call'}
PROPERTY PUBLIC msgSevyIsWarning : BOOL
GET
msgSevyIsWarning := MsgSeverity = 1;
END_GET
END_PROPERTY

END_FUNCTION_BLOCK

